(*Deactivate*)
ARsDeactivateDescription	[172]		:=		'[ DA-0172 ] OutputSignal - Reserved';
ARbDeactivateOutput		[172]		:=		FALSE or ARbDeactivateTestPB[172];

(*Deactivate*)
ARsDeactivateDescription	[173]		:=		'[ DA-0173 ] OutputSignal - Reserved';
ARbDeactivateOutput		[173]		:=		FALSE or ARbDeactivateTestPB[173];

(*Deactivate*)
ARsDeactivateDescription	[174]		:=		'[ DA-0174 ] OutputSignal - Reserved';
ARbDeactivateOutput		[174]		:=		FALSE or ARbDeactivateTestPB[174];

(*Deactivate*)
ARsDeactivateDescription	[175]		:=		'[ DA-0175 ] OutputSignal - Reserved';
ARbDeactivateOutput		[175]		:=		FALSE or ARbDeactivateTestPB[175];

(*Deactivate*)
ARsDeactivateDescription	[176]		:=		'[ DA-0176 ] OutputSignal - Reserved';
ARbDeactivateOutput		[176]		:=		FALSE or ARbDeactivateTestPB[176];

(*Deactivate*)
ARsDeactivateDescription	[177]		:=		'[ DA-0177 ] OutputSignal - Reserved';
ARbDeactivateOutput		[177]		:=		FALSE or ARbDeactivateTestPB[177];

(*Deactivate*)
ARsDeactivateDescription	[178]		:=		'[ DA-0178 ] OutputSignal - Reserved';
ARbDeactivateOutput		[178]		:=		FALSE or ARbDeactivateTestPB[178];

(*Deactivate*)
ARsDeactivateDescription	[179]		:=		'[ DA-0179 ] OutputSignal - Reserved';
ARbDeactivateOutput		[179]		:=		FALSE or ARbDeactivateTestPB[179];

(*Deactivate*)
ARsDeactivateDescription	[180]		:=		'[ DA-0180 ] OutputSignal - Reserved';
ARbDeactivateOutput		[180]		:=		FALSE or ARbDeactivateTestPB[180];

(*Deactivate*)
ARsDeactivateDescription	[181]		:=		'[ DA-0181 ] OutputSignal - Reserved';
ARbDeactivateOutput		[181]		:=		FALSE or ARbDeactivateTestPB[181];

(*Deactivate*)
ARsDeactivateDescription	[182]		:=		'[ DA-0182 ] OutputSignal - Reserved';
ARbDeactivateOutput		[182]		:=		FALSE or ARbDeactivateTestPB[182];

(*Deactivate*)
ARsDeactivateDescription	[183]		:=		'[ DA-0183 ] OutputSignal - Reserved';
ARbDeactivateOutput		[183]		:=		FALSE or ARbDeactivateTestPB[183];

(*Deactivate*)
ARsDeactivateDescription	[184]		:=		'[ DA-0184 ] OutputSignal - Reserved';
ARbDeactivateOutput		[184]		:=		FALSE or ARbDeactivateTestPB[184];

(*Deactivate*)
ARsDeactivateDescription	[185]		:=		'[ DA-0185 ] OutputSignal - Reserved';
ARbDeactivateOutput		[185]		:=		FALSE or ARbDeactivateTestPB[185];

(*Deactivate*)
ARsDeactivateDescription	[186]		:=		'[ DA-0186 ] OutputSignal - Reserved';
ARbDeactivateOutput		[186]		:=		FALSE or ARbDeactivateTestPB[186];

(*Deactivate*)
ARsDeactivateDescription	[187]		:=		'[ DA-0187 ] OutputSignal - Reserved';
ARbDeactivateOutput		[187]		:=		FALSE or ARbDeactivateTestPB[187];

(*Deactivate*)
ARsDeactivateDescription	[188]		:=		'[ DA-0188 ] OutputSignal - Reserved';
ARbDeactivateOutput		[188]		:=		FALSE or ARbDeactivateTestPB[188];

(*Deactivate*)
ARsDeactivateDescription	[189]		:=		'[ DA-0189 ] OutputSignal - Reserved';
ARbDeactivateOutput		[189]		:=		FALSE or ARbDeactivateTestPB[189];

(*Deactivate*)
ARsDeactivateDescription	[190]		:=		'[ DA-0190 ] OutputSignal - Reserved';
ARbDeactivateOutput		[190]		:=		FALSE or ARbDeactivateTestPB[190];

(*Deactivate*)
ARsDeactivateDescription	[191]		:=		'[ DA-0191 ] OutputSignal - Reserved';
ARbDeactivateOutput		[191]		:=		FALSE or ARbDeactivateTestPB[191];

(*Deactivate*)
ARsDeactivateDescription	[192]		:=		'[ DA-0192 ] OutputSignal - Reserved';
ARbDeactivateOutput		[192]		:=		FALSE or ARbDeactivateTestPB[192];

(*Deactivate*)
ARsDeactivateDescription	[193]		:=		'[ DA-0193 ] OutputSignal - Reserved';
ARbDeactivateOutput		[193]		:=		FALSE or ARbDeactivateTestPB[193];

(*Deactivate*)
ARsDeactivateDescription	[194]		:=		'[ DA-0194 ] OutputSignal - Reserved';
ARbDeactivateOutput		[194]		:=		FALSE or ARbDeactivateTestPB[194];

(*Deactivate*)
ARsDeactivateDescription	[195]		:=		'[ DA-0195 ] OutputSignal - Reserved';
ARbDeactivateOutput		[195]		:=		FALSE or ARbDeactivateTestPB[195];

(*Deactivate*)
ARsDeactivateDescription	[196]		:=		'[ DA-0196 ] OutputSignal - Reserved';
ARbDeactivateOutput		[196]		:=		FALSE or ARbDeactivateTestPB[196];

(*Deactivate*)
ARsDeactivateDescription	[197]		:=		'[ DA-0197 ] OutputSignal - Reserved';
ARbDeactivateOutput		[197]		:=		FALSE or ARbDeactivateTestPB[197];

(*Deactivate*)
ARsDeactivateDescription	[198]		:=		'[ DA-0198 ] OutputSignal - Reserved';
ARbDeactivateOutput		[198]		:=		FALSE or ARbDeactivateTestPB[198];

(*Deactivate*)
ARsDeactivateDescription	[199]		:=		'[ DA-0199 ] OutputSignal - Reserved';
ARbDeactivateOutput		[199]		:=		FALSE or ARbDeactivateTestPB[199];

(*Deactivate*)
ARsDeactivateDescription	[200]		:=		'[ DA-0200 ] OutputSignal - Reserved';
ARbDeactivateOutput		[200]		:=		FALSE or ARbDeactivateTestPB[200];
*)
*)

END_PROGRAM

// ---- POUs/MainProgram/AutoArmCtrl/OmronServoEnable.TcPOU
PROGRAM OmronServoEnable
VAR
END_VAR

IF PowerOnDelay.Q AND NOT EmergencyStop THEN
	ARwDO[eY10007_STN09SLOWPULLMECHANISMSERVOMOTOR_ERRORSTOP].00 := TRUE;
	ARwDO[eY10008_Arm01HorizontalServoMotor_ErrorStop].00 := TRUE;
	ARwDO[eY10009_Arm01VerticalServoMotor_ErrorStop].00 := TRUE;
	ELSE
	ARwDO[eY10007_STN09SLOWPULLMECHANISMSERVOMOTOR_ERRORSTOP].00 := FALSE;
	ARwDO[eY10008_Arm01HorizontalServoMotor_ErrorStop].00 := FALSE;
	ARwDO[eY10009_Arm01VerticalServoMotor_ErrorStop].00 := FALSE;
END_IF

END_PROGRAM

// ---- POUs/MainProgram/AutoArmCtrl/AxisHorzMovementOutputCtrl_Arm1.TcPOU
PROGRAM AxisHorzMovementOutputCtrl_Arm1
VAR

	LdUnhook: CMP_OC_DW;
	Stn1Unhook: CMP_OC_DW;
	Stn2Unhook: CMP_OC_DW;
	Stn3Unhook: CMP_OC_DW;
	Stn4Unhook: CMP_OC_DW;
	Stn5Unhook: CMP_OC_DW;
	Stn6Unhook: CMP_OC_DW;
	Stn7Unhook: CMP_OC_DW;
	Stn8Unhook: CMP_OC_DW;
	Stn9Unhook: CMP_OC_DW;
	Stn10Unhook: CMP_OC_DW;
	Stn11Unhook: CMP_OC_DW;
	Stn12Unhook: CMP_OC_DW;
	Uld1Unhook: CMP_OC_DW;
	Uld2Unhook: CMP_OC_DW;

	LdHook: CMP_OC_DW;
	Stn1Hook: CMP_OC_DW;
	Stn2Hook: CMP_OC_DW;
	Stn3Hook: CMP_OC_DW;
	Stn4Hook: CMP_OC_DW;
	Stn5Hook: CMP_OC_DW;
	Stn6Hook: CMP_OC_DW;
	Stn7Hook: CMP_OC_DW;
	Stn8Hook: CMP_OC_DW;
	Stn9Hook: CMP_OC_DW;
	Stn10Hook: CMP_OC_DW;
	Stn11Hook: CMP_OC_DW;
	Stn12Hook: CMP_OC_DW;
	Uld1Hook: CMP_OC_DW;
	Uld2Hook: CMP_OC_DW;

END_VAR

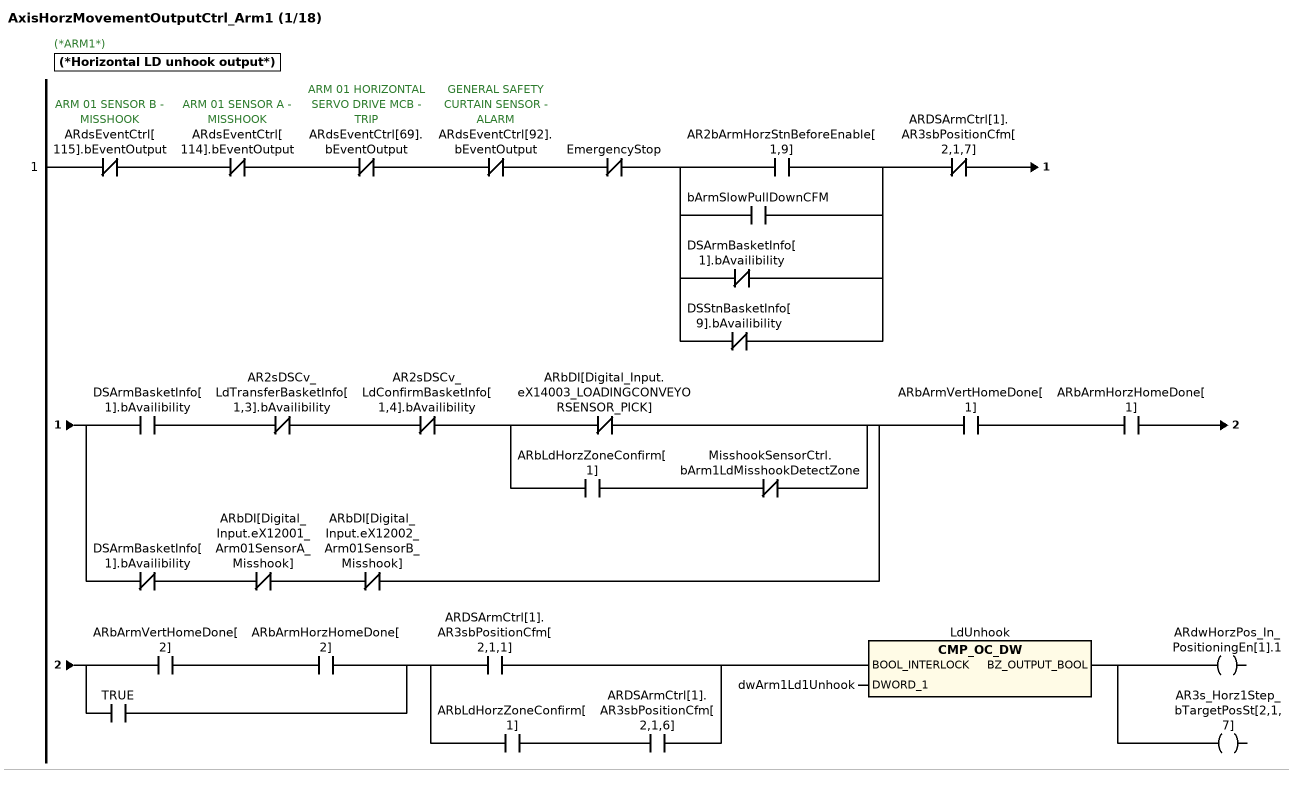
// NETWORK 1
// (*ARM1*)
//   ARdsEventCtrl[115].bEventOutput: ARM 01 SENSOR B - MISSHOOK
//   ARdsEventCtrl[114].bEventOutput: ARM 01 SENSOR A - MISSHOOK
//   ARdsEventCtrl[69].bEventOutput: ARM 01 HORIZONTAL SERVO DRIVE MCB - TRIP
//   ARdsEventCtrl[92].bEventOutput: GENERAL SAFETY CURTAIN SENSOR - ALARM
// label: (*Horizontal LD unhook output*)
LdUnhook(BOOL_INTERLOCK := (((NOT ARdsEventCtrl[115].bEventOutput AND NOT ARdsEventCtrl[114].bEventOutput AND NOT ARdsEventCtrl[69].bEventOutput AND NOT ARdsEventCtrl[92].bEventOutput AND NOT EmergencyStop) AND (AR2bArmHorzStnBeforeEnable[1,9] OR bArmSlowPullDownCFM OR NOT DSArmBasketInfo[1].bAvailibility OR NOT DSStnBasketInfo[9].bAvailibility)) AND NOT ARDSArmCtrl[1].AR3sbPositionCfm[2,1,7] AND (DSArmBasketInfo[1].bAvailibility AND NOT AR2sDSCv_LdTransferBasketInfo[1,3].bAvailibility AND NOT AR2sDSCv_LdConfirmBasketInfo[1,4].bAvailibility AND (NOT ARbDI[Digital_Input.eX14003_LOADINGCONVEYORSENSOR_PICK] OR ARbLdHorzZoneConfirm[1] AND NOT MisshookSensorCtrl.bArm1LdMisshookDetectZone) OR NOT DSArmBasketInfo[1].bAvailibility AND NOT ARbDI[Digital_Input.eX12001_Arm01SensorA_Misshook] AND NOT ARbDI[Digital_Input.eX12002_Arm01SensorB_Misshook])) AND ARbArmVertHomeDone[1] AND ARbArmHorzHomeDone[1] AND (ARbArmVertHomeDone[2] AND ARbArmHorzHomeDone[2] OR TRUE) AND (ARDSArmCtrl[1].AR3sbPositionCfm[2,1,1] OR ARbLdHorzZoneConfirm[1] AND ARDSArmCtrl[1].AR3sbPositionCfm[2,1,6]), DWORD_1 := dwArm1Ld1Unhook); // CMP_OC_DW
ARdwHorzPos_In_PositioningEn[1].1 := LdUnhook.BZ_OUTPUT_BOOL;
AR3s_Horz1Step_bTargetPosSt[2,1,7] := LdUnhook.BZ_OUTPUT_BOOL;

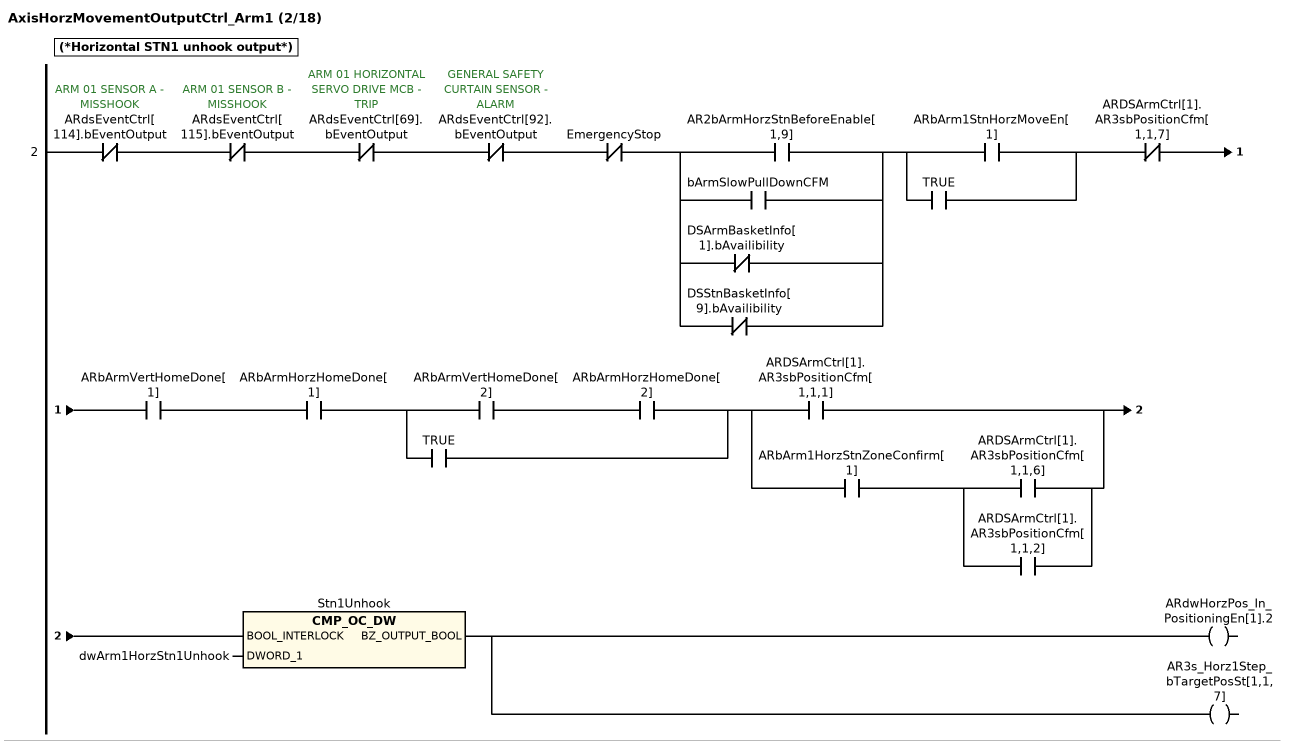
// NETWORK 2
//   ARdsEventCtrl[114].bEventOutput: ARM 01 SENSOR A - MISSHOOK
//   ARdsEventCtrl[115].bEventOutput: ARM 01 SENSOR B - MISSHOOK
//   ARdsEventCtrl[69].bEventOutput: ARM 01 HORIZONTAL SERVO DRIVE MCB - TRIP
//   ARdsEventCtrl[92].bEventOutput: GENERAL SAFETY CURTAIN SENSOR - ALARM
// label: (*Horizontal STN1 unhook output*)
Stn1Unhook(BOOL_INTERLOCK := ((NOT ARdsEventCtrl[114].bEventOutput AND NOT ARdsEventCtrl[115].bEventOutput AND NOT ARdsEventCtrl[69].bEventOutput AND NOT ARdsEventCtrl[92].bEventOutput AND NOT EmergencyStop) AND (AR2bArmHorzStnBeforeEnable[1,9] OR bArmSlowPullDownCFM OR NOT DSArmBasketInfo[1].bAvailibility OR NOT DSStnBasketInfo[9].bAvailibility) AND (ARbArm1StnHorzMoveEn[1] OR TRUE)) AND NOT ARDSArmCtrl[1].AR3sbPositionCfm[1,1,7] AND ARbArmVertHomeDone[1] AND ARbArmHorzHomeDone[1] AND (ARbArmVertHomeDone[2] AND ARbArmHorzHomeDone[2] OR TRUE) AND (ARDSArmCtrl[1].AR3sbPositionCfm[1,1,1] OR ARbArm1HorzStnZoneConfirm[1] AND (ARDSArmCtrl[1].AR3sbPositionCfm[1,1,6] OR ARDSArmCtrl[1].AR3sbPositionCfm[1,1,2])), DWORD_1 := dwArm1HorzStn1Unhook); // CMP_OC_DW
ARdwHorzPos_In_PositioningEn[1].2 := Stn1Unhook.BZ_OUTPUT_BOOL;
AR3s_Horz1Step_bTargetPosSt[1,1,7] := Stn1Unhook.BZ_OUTPUT_BOOL;

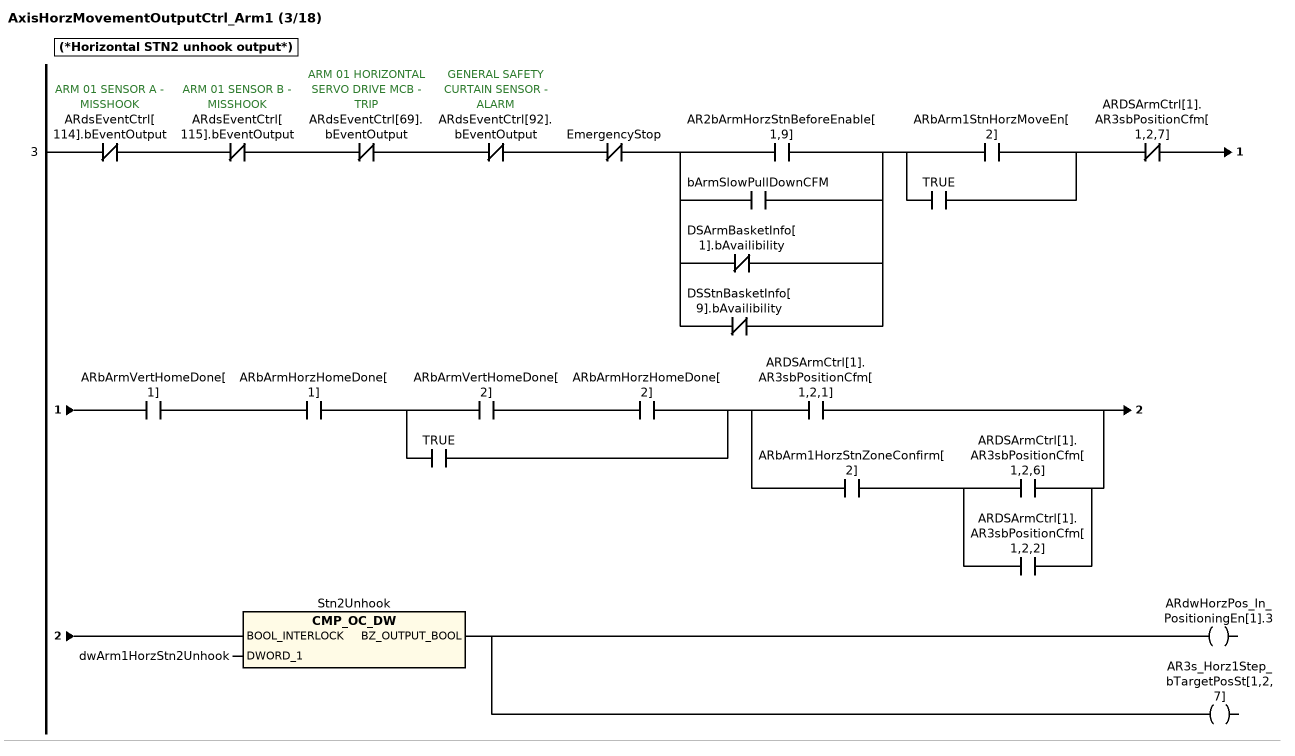
// NETWORK 3
//   ARdsEventCtrl[114].bEventOutput: ARM 01 SENSOR A - MISSHOOK
//   ARdsEventCtrl[115].bEventOutput: ARM 01 SENSOR B - MISSHOOK
//   ARdsEventCtrl[69].bEventOutput: ARM 01 HORIZONTAL SERVO DRIVE MCB - TRIP
//   ARdsEventCtrl[92].bEventOutput: GENERAL SAFETY CURTAIN SENSOR - ALARM
// label: (*Horizontal STN2 unhook output*)
Stn2Unhook(BOOL_INTERLOCK := ((NOT ARdsEventCtrl[114].bEventOutput AND NOT ARdsEventCtrl[115].bEventOutput AND NOT ARdsEventCtrl[69].bEventOutput AND NOT ARdsEventCtrl[92].bEventOutput AND NOT EmergencyStop) AND (AR2bArmHorzStnBeforeEnable[1,9] OR bArmSlowPullDownCFM OR NOT DSArmBasketInfo[1].bAvailibility OR NOT DSStnBasketInfo[9].bAvailibility) AND (ARbArm1StnHorzMoveEn[2] OR TRUE)) AND NOT ARDSArmCtrl[1].AR3sbPositionCfm[1,2,7] AND ARbArmVertHomeDone[1] AND ARbArmHorzHomeDone[1] AND (ARbArmVertHomeDone[2] AND ARbArmHorzHomeDone[2] OR TRUE) AND (ARDSArmCtrl[1].AR3sbPositionCfm[1,2,1] OR ARbArm1HorzStnZoneConfirm[2] AND (ARDSArmCtrl[1].AR3sbPositionCfm[1,2,6] OR ARDSArmCtrl[1].AR3sbPositionCfm[1,2,2])), DWORD_1 := dwArm1HorzStn2Unhook); // CMP_OC_DW
ARdwHorzPos_In_PositioningEn[1].3 := Stn2Unhook.BZ_OUTPUT_BOOL;
AR3s_Horz1Step_bTargetPosSt[1,2,7] := Stn2Unhook.BZ_OUTPUT_BOOL;

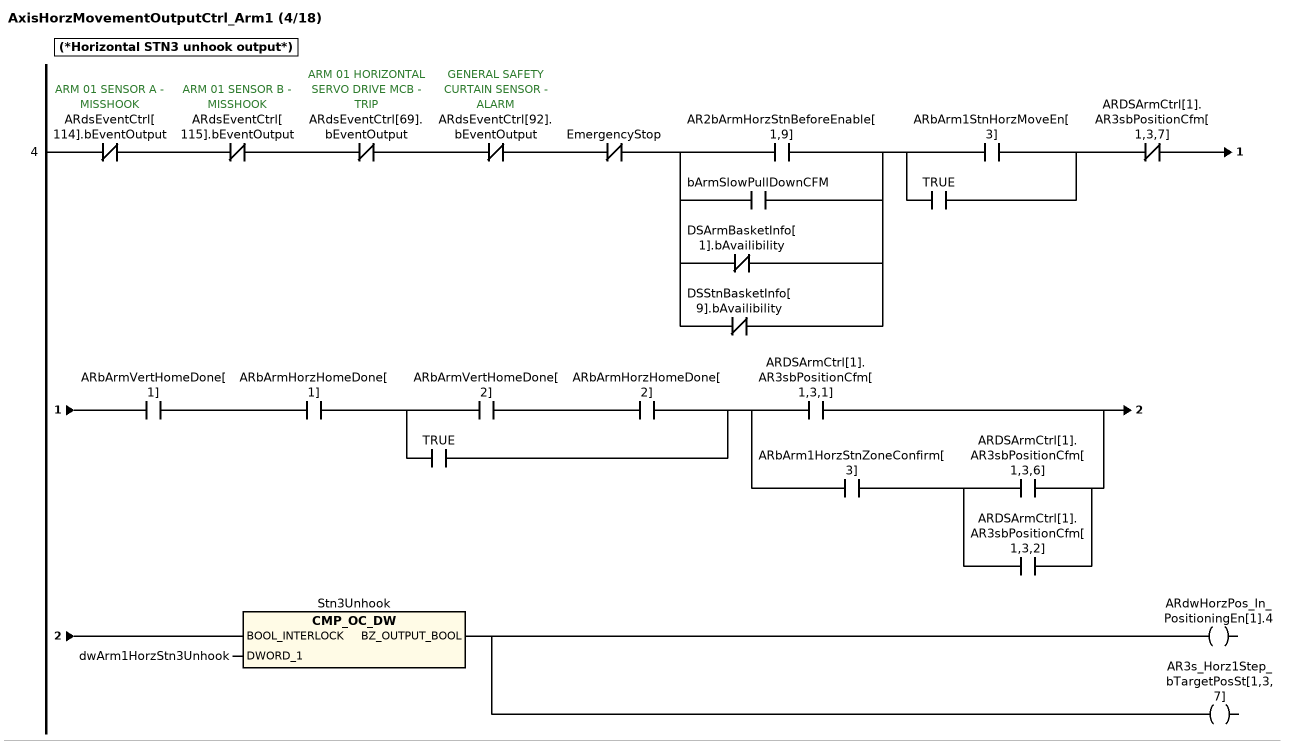
// NETWORK 4
//   ARdsEventCtrl[114].bEventOutput: ARM 01 SENSOR A - MISSHOOK
//   ARdsEventCtrl[115].bEventOutput: ARM 01 SENSOR B - MISSHOOK
//   ARdsEventCtrl[69].bEventOutput: ARM 01 HORIZONTAL SERVO DRIVE MCB - TRIP
//   ARdsEventCtrl[92].bEventOutput: GENERAL SAFETY CURTAIN SENSOR - ALARM
// label: (*Horizontal STN3 unhook output*)
Stn3Unhook(BOOL_INTERLOCK := ((NOT ARdsEventCtrl[114].bEventOutput AND NOT ARdsEventCtrl[115].bEventOutput AND NOT ARdsEventCtrl[69].bEventOutput AND NOT ARdsEventCtrl[92].bEventOutput AND NOT EmergencyStop) AND (AR2bArmHorzStnBeforeEnable[1,9] OR bArmSlowPullDownCFM OR NOT DSArmBasketInfo[1].bAvailibility OR NOT DSStnBasketInfo[9].bAvailibility) AND (ARbArm1StnHorzMoveEn[3] OR TRUE)) AND NOT ARDSArmCtrl[1].AR3sbPositionCfm[1,3,7] AND ARbArmVertHomeDone[1] AND ARbArmHorzHomeDone[1] AND (ARbArmVertHomeDone[2] AND ARbArmHorzHomeDone[2] OR TRUE) AND (ARDSArmCtrl[1].AR3sbPositionCfm[1,3,1] OR ARbArm1HorzStnZoneConfirm[3] AND (ARDSArmCtrl[1].AR3sbPositionCfm[1,3,6] OR ARDSArmCtrl[1].AR3sbPositionCfm[1,3,2])), DWORD_1 := dwArm1HorzStn3Unhook); // CMP_OC_DW
ARdwHorzPos_In_PositioningEn[1].4 := Stn3Unhook.BZ_OUTPUT_BOOL;
AR3s_Horz1Step_bTargetPosSt[1,3,7] := Stn3Unhook.BZ_OUTPUT_BOOL;

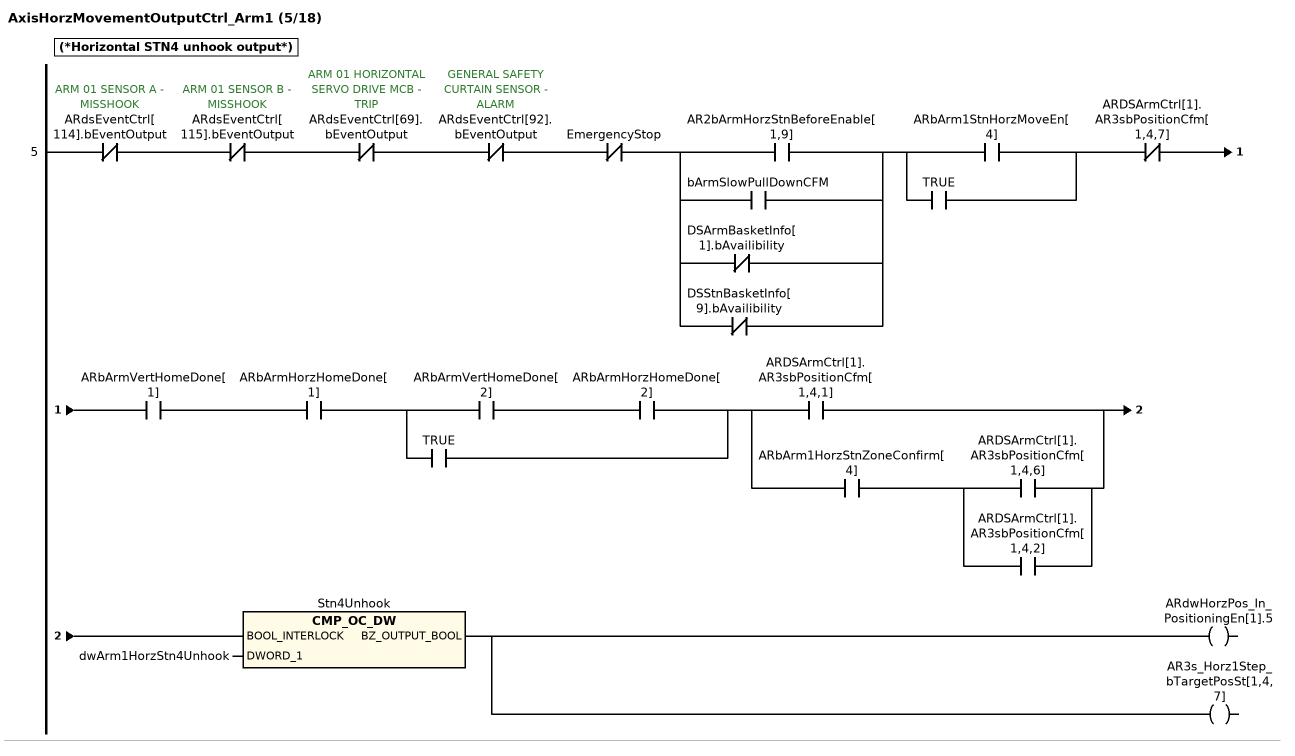
// NETWORK 5
//   ARdsEventCtrl[114].bEventOutput: ARM 01 SENSOR A - MISSHOOK
//   ARdsEventCtrl[115].bEventOutput: ARM 01 SENSOR B - MISSHOOK
//   ARdsEventCtrl[69].bEventOutput: ARM 01 HORIZONTAL SERVO DRIVE MCB - TRIP
//   ARdsEventCtrl[92].bEventOutput: GENERAL SAFETY CURTAIN SENSOR - ALARM
// label: (*Horizontal STN4 unhook output*)
Stn4Unhook(BOOL_INTERLOCK := ((NOT ARdsEventCtrl[114].bEventOutput AND NOT ARdsEventCtrl[115].bEventOutput AND NOT ARdsEventCtrl[69].bEventOutput AND NOT ARdsEventCtrl[92].bEventOutput AND NOT EmergencyStop) AND (AR2bArmHorzStnBeforeEnable[1,9] OR bArmSlowPullDownCFM OR NOT DSArmBasketInfo[1].bAvailibility OR NOT DSStnBasketInfo[9].bAvailibility) AND (ARbArm1StnHorzMoveEn[4] OR TRUE)) AND NOT ARDSArmCtrl[1].AR3sbPositionCfm[1,4,7] AND ARbArmVertHomeDone[1] AND ARbArmHorzHomeDone[1] AND (ARbArmVertHomeDone[2] AND ARbArmHorzHomeDone[2] OR TRUE) AND (ARDSArmCtrl[1].AR3sbPositionCfm[1,4,1] OR ARbArm1HorzStnZoneConfirm[4] AND (ARDSArmCtrl[1].AR3sbPositionCfm[1,4,6] OR ARDSArmCtrl[1].AR3sbPositionCfm[1,4,2])), DWORD_1 := dwArm1HorzStn4Unhook); // CMP_OC_DW
ARdwHorzPos_In_PositioningEn[1].5 := Stn4Unhook.BZ_OUTPUT_BOOL;
AR3s_Horz1Step_bTargetPosSt[1,4,7] := Stn4Unhook.BZ_OUTPUT_BOOL;

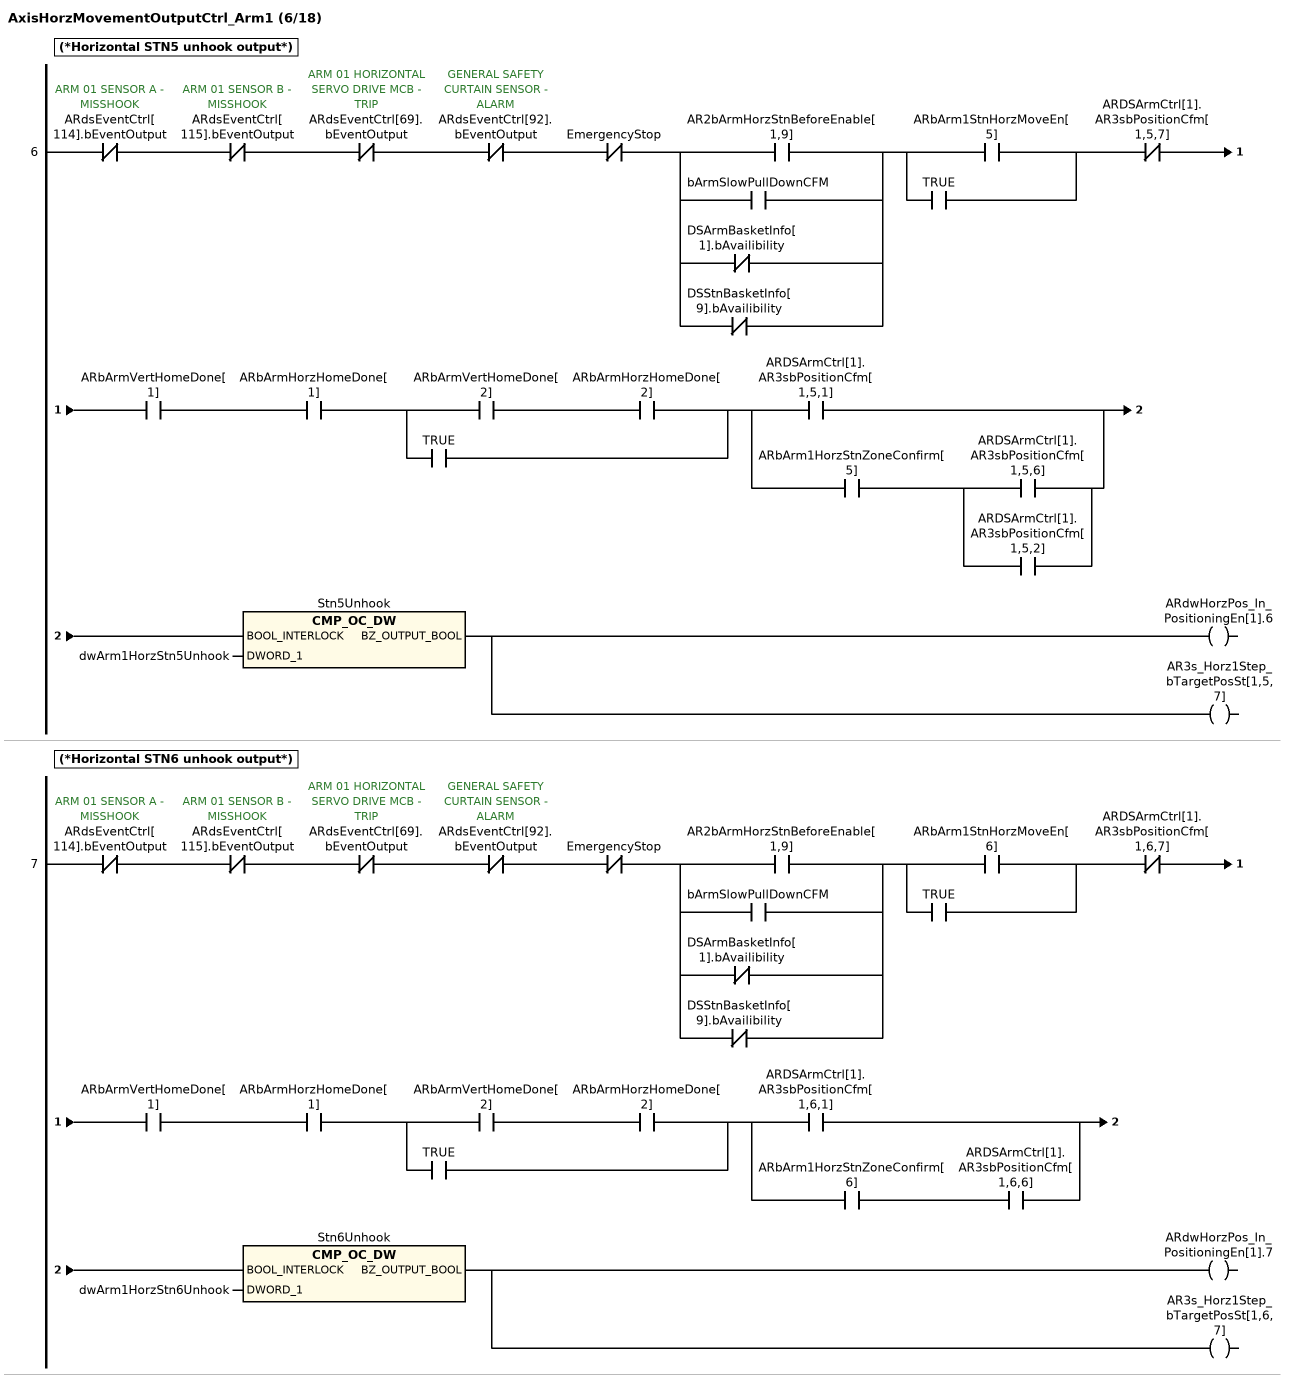
// NETWORK 6
//   ARdsEventCtrl[114].bEventOutput: ARM 01 SENSOR A - MISSHOOK
//   ARdsEventCtrl[115].bEventOutput: ARM 01 SENSOR B - MISSHOOK
//   ARdsEventCtrl[69].bEventOutput: ARM 01 HORIZONTAL SERVO DRIVE MCB - TRIP
//   ARdsEventCtrl[92].bEventOutput: GENERAL SAFETY CURTAIN SENSOR - ALARM
// label: (*Horizontal STN5 unhook output*)
Stn5Unhook(BOOL_INTERLOCK := ((NOT ARdsEventCtrl[114].bEventOutput AND NOT ARdsEventCtrl[115].bEventOutput AND NOT ARdsEventCtrl[69].bEventOutput AND NOT ARdsEventCtrl[92].bEventOutput AND NOT EmergencyStop) AND (AR2bArmHorzStnBeforeEnable[1,9] OR bArmSlowPullDownCFM OR NOT DSArmBasketInfo[1].bAvailibility OR NOT DSStnBasketInfo[9].bAvailibility) AND (ARbArm1StnHorzMoveEn[5] OR TRUE)) AND NOT ARDSArmCtrl[1].AR3sbPositionCfm[1,5,7] AND ARbArmVertHomeDone[1] AND ARbArmHorzHomeDone[1] AND (ARbArmVertHomeDone[2] AND ARbArmHorzHomeDone[2] OR TRUE) AND (ARDSArmCtrl[1].AR3sbPositionCfm[1,5,1] OR ARbArm1HorzStnZoneConfirm[5] AND (ARDSArmCtrl[1].AR3sbPositionCfm[1,5,6] OR ARDSArmCtrl[1].AR3sbPositionCfm[1,5,2])), DWORD_1 := dwArm1HorzStn5Unhook); // CMP_OC_DW
ARdwHorzPos_In_PositioningEn[1].6 := Stn5Unhook.BZ_OUTPUT_BOOL;
AR3s_Horz1Step_bTargetPosSt[1,5,7] := Stn5Unhook.BZ_OUTPUT_BOOL;

// NETWORK 7
//   ARdsEventCtrl[114].bEventOutput: ARM 01 SENSOR A - MISSHOOK
//   ARdsEventCtrl[115].bEventOutput: ARM 01 SENSOR B - MISSHOOK
//   ARdsEventCtrl[69].bEventOutput: ARM 01 HORIZONTAL SERVO DRIVE MCB - TRIP
//   ARdsEventCtrl[92].bEventOutput: GENERAL SAFETY CURTAIN SENSOR - ALARM
// label: (*Horizontal STN6 unhook output*)
Stn6Unhook(BOOL_INTERLOCK := ((NOT ARdsEventCtrl[114].bEventOutput AND NOT ARdsEventCtrl[115].bEventOutput AND NOT ARdsEventCtrl[69].bEventOutput AND NOT ARdsEventCtrl[92].bEventOutput AND NOT EmergencyStop) AND ((AR2bArmHorzStnBeforeEnable[1,9] OR bArmSlowPullDownCFM OR NOT DSArmBasketInfo[1].bAvailibility OR NOT DSStnBasketInfo[9].bAvailibility) AND (ARbArm1StnHorzMoveEn[6] OR TRUE))) AND NOT ARDSArmCtrl[1].AR3sbPositionCfm[1,6,7] AND ARbArmVertHomeDone[1] AND ARbArmHorzHomeDone[1] AND (ARbArmVertHomeDone[2] AND ARbArmHorzHomeDone[2] OR TRUE) AND (ARDSArmCtrl[1].AR3sbPositionCfm[1,6,1] OR ARbArm1HorzStnZoneConfirm[6] AND ARDSArmCtrl[1].AR3sbPositionCfm[1,6,6]), DWORD_1 := dwArm1HorzStn6Unhook); // CMP_OC_DW
ARdwHorzPos_In_PositioningEn[1].7 := Stn6Unhook.BZ_OUTPUT_BOOL;
AR3s_Horz1Step_bTargetPosSt[1,6,7] := Stn6Unhook.BZ_OUTPUT_BOOL;

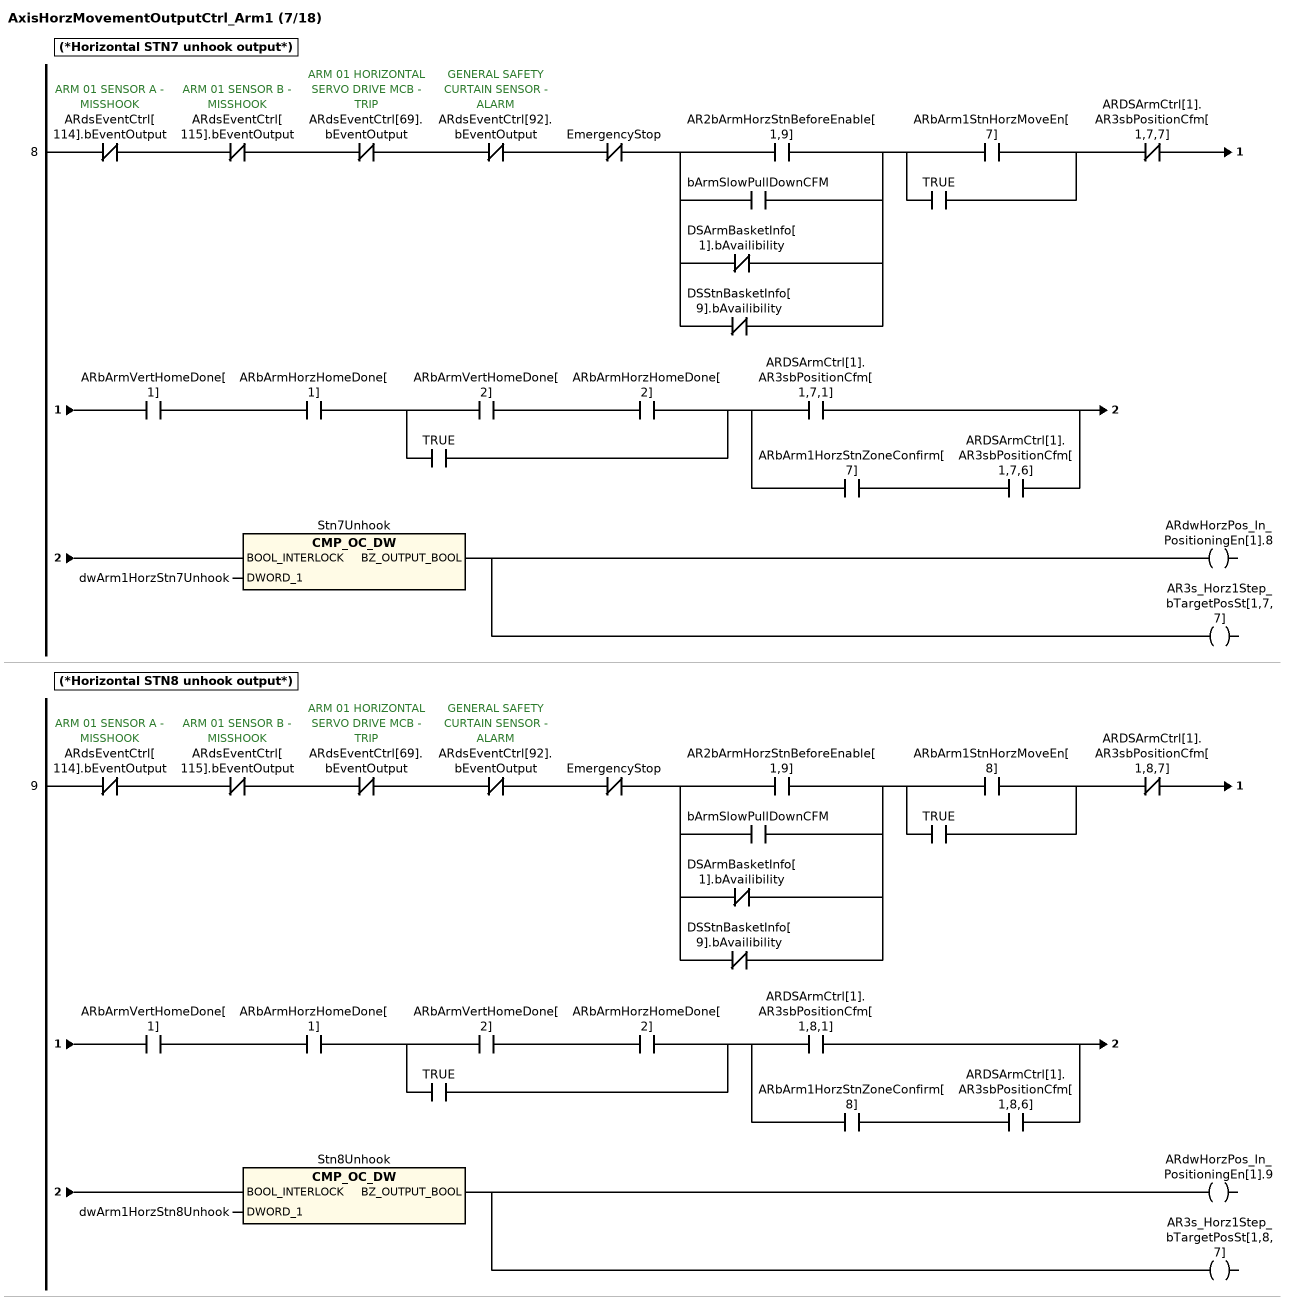
// NETWORK 8
//   ARdsEventCtrl[114].bEventOutput: ARM 01 SENSOR A - MISSHOOK
//   ARdsEventCtrl[115].bEventOutput: ARM 01 SENSOR B - MISSHOOK
//   ARdsEventCtrl[69].bEventOutput: ARM 01 HORIZONTAL SERVO DRIVE MCB - TRIP
//   ARdsEventCtrl[92].bEventOutput: GENERAL SAFETY CURTAIN SENSOR - ALARM
// label: (*Horizontal STN7 unhook output*)
Stn7Unhook(BOOL_INTERLOCK := ((NOT ARdsEventCtrl[114].bEventOutput AND NOT ARdsEventCtrl[115].bEventOutput AND NOT ARdsEventCtrl[69].bEventOutput AND NOT ARdsEventCtrl[92].bEventOutput AND NOT EmergencyStop) AND (AR2bArmHorzStnBeforeEnable[1,9] OR bArmSlowPullDownCFM OR NOT DSArmBasketInfo[1].bAvailibility OR NOT DSStnBasketInfo[9].bAvailibility) AND (ARbArm1StnHorzMoveEn[7] OR TRUE)) AND NOT ARDSArmCtrl[1].AR3sbPositionCfm[1,7,7] AND ARbArmVertHomeDone[1] AND ARbArmHorzHomeDone[1] AND (ARbArmVertHomeDone[2] AND ARbArmHorzHomeDone[2] OR TRUE) AND (ARDSArmCtrl[1].AR3sbPositionCfm[1,7,1] OR ARbArm1HorzStnZoneConfirm[7] AND ARDSArmCtrl[1].AR3sbPositionCfm[1,7,6]), DWORD_1 := dwArm1HorzStn7Unhook); // CMP_OC_DW
ARdwHorzPos_In_PositioningEn[1].8 := Stn7Unhook.BZ_OUTPUT_BOOL;
AR3s_Horz1Step_bTargetPosSt[1,7,7] := Stn7Unhook.BZ_OUTPUT_BOOL;

// NETWORK 9
//   ARdsEventCtrl[114].bEventOutput: ARM 01 SENSOR A - MISSHOOK
//   ARdsEventCtrl[115].bEventOutput: ARM 01 SENSOR B - MISSHOOK
//   ARdsEventCtrl[69].bEventOutput: ARM 01 HORIZONTAL SERVO DRIVE MCB - TRIP
//   ARdsEventCtrl[92].bEventOutput: GENERAL SAFETY CURTAIN SENSOR - ALARM
// label: (*Horizontal STN8 unhook output*)
Stn8Unhook(BOOL_INTERLOCK := ((NOT ARdsEventCtrl[114].bEventOutput AND NOT ARdsEventCtrl[115].bEventOutput AND NOT ARdsEventCtrl[69].bEventOutput AND NOT ARdsEventCtrl[92].bEventOutput AND NOT EmergencyStop) AND (AR2bArmHorzStnBeforeEnable[1,9] OR bArmSlowPullDownCFM OR NOT DSArmBasketInfo[1].bAvailibility OR NOT DSStnBasketInfo[9].bAvailibility) AND (ARbArm1StnHorzMoveEn[8] OR TRUE)) AND NOT ARDSArmCtrl[1].AR3sbPositionCfm[1,8,7] AND ARbArmVertHomeDone[1] AND ARbArmHorzHomeDone[1] AND (ARbArmVertHomeDone[2] AND ARbArmHorzHomeDone[2] OR TRUE) AND (ARDSArmCtrl[1].AR3sbPositionCfm[1,8,1] OR ARbArm1HorzStnZoneConfirm[8] AND ARDSArmCtrl[1].AR3sbPositionCfm[1,8,6]), DWORD_1 := dwArm1HorzStn8Unhook); // CMP_OC_DW
ARdwHorzPos_In_PositioningEn[1].9 := Stn8Unhook.BZ_OUTPUT_BOOL;
AR3s_Horz1Step_bTargetPosSt[1,8,7] := Stn8Unhook.BZ_OUTPUT_BOOL;

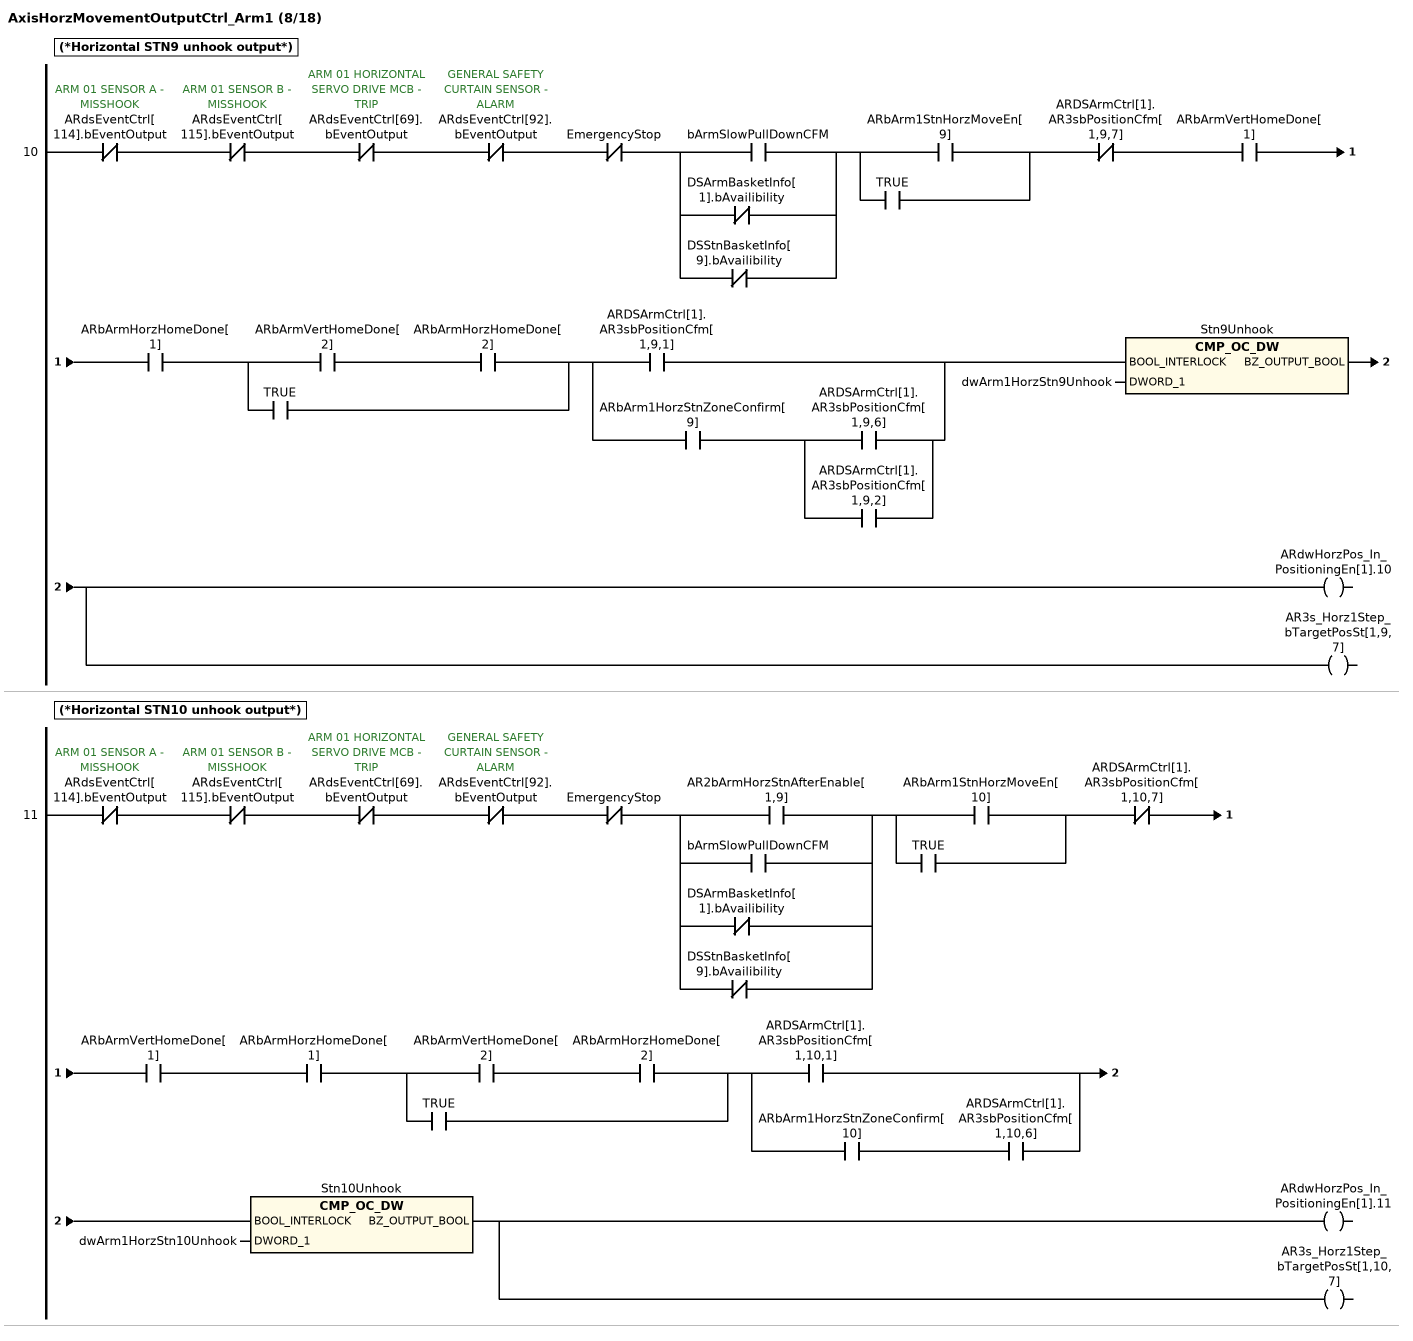
// NETWORK 10
//   ARdsEventCtrl[114].bEventOutput: ARM 01 SENSOR A - MISSHOOK
//   ARdsEventCtrl[115].bEventOutput: ARM 01 SENSOR B - MISSHOOK
//   ARdsEventCtrl[69].bEventOutput: ARM 01 HORIZONTAL SERVO DRIVE MCB - TRIP
//   ARdsEventCtrl[92].bEventOutput: GENERAL SAFETY CURTAIN SENSOR - ALARM
// label: (*Horizontal STN9 unhook output*)
Stn9Unhook(BOOL_INTERLOCK := ((NOT ARdsEventCtrl[114].bEventOutput AND NOT ARdsEventCtrl[115].bEventOutput AND NOT ARdsEventCtrl[69].bEventOutput AND NOT ARdsEventCtrl[92].bEventOutput AND NOT EmergencyStop) AND (bArmSlowPullDownCFM OR NOT DSArmBasketInfo[1].bAvailibility OR NOT DSStnBasketInfo[9].bAvailibility) AND (ARbArm1StnHorzMoveEn[9] OR TRUE)) AND NOT ARDSArmCtrl[1].AR3sbPositionCfm[1,9,7] AND ARbArmVertHomeDone[1] AND ARbArmHorzHomeDone[1] AND (ARbArmVertHomeDone[2] AND ARbArmHorzHomeDone[2] OR TRUE) AND (ARDSArmCtrl[1].AR3sbPositionCfm[1,9,1] OR ARbArm1HorzStnZoneConfirm[9] AND (ARDSArmCtrl[1].AR3sbPositionCfm[1,9,6] OR ARDSArmCtrl[1].AR3sbPositionCfm[1,9,2])), DWORD_1 := dwArm1HorzStn9Unhook); // CMP_OC_DW
ARdwHorzPos_In_PositioningEn[1].10 := Stn9Unhook.BZ_OUTPUT_BOOL;
AR3s_Horz1Step_bTargetPosSt[1,9,7] := Stn9Unhook.BZ_OUTPUT_BOOL;

// NETWORK 11
//   ARdsEventCtrl[114].bEventOutput: ARM 01 SENSOR A - MISSHOOK
//   ARdsEventCtrl[115].bEventOutput: ARM 01 SENSOR B - MISSHOOK
//   ARdsEventCtrl[69].bEventOutput: ARM 01 HORIZONTAL SERVO DRIVE MCB - TRIP
//   ARdsEventCtrl[92].bEventOutput: GENERAL SAFETY CURTAIN SENSOR - ALARM
// label: (*Horizontal STN10 unhook output*)
Stn10Unhook(BOOL_INTERLOCK := ((NOT ARdsEventCtrl[114].bEventOutput AND NOT ARdsEventCtrl[115].bEventOutput AND NOT ARdsEventCtrl[69].bEventOutput AND NOT ARdsEventCtrl[92].bEventOutput AND NOT EmergencyStop) AND (AR2bArmHorzStnAfterEnable[1,9] OR bArmSlowPullDownCFM OR NOT DSArmBasketInfo[1].bAvailibility OR NOT DSStnBasketInfo[9].bAvailibility) AND (ARbArm1StnHorzMoveEn[10] OR TRUE)) AND NOT ARDSArmCtrl[1].AR3sbPositionCfm[1,10,7] AND ARbArmVertHomeDone[1] AND ARbArmHorzHomeDone[1] AND (ARbArmVertHomeDone[2] AND ARbArmHorzHomeDone[2] OR TRUE) AND (ARDSArmCtrl[1].AR3sbPositionCfm[1,10,1] OR ARbArm1HorzStnZoneConfirm[10] AND ARDSArmCtrl[1].AR3sbPositionCfm[1,10,6]), DWORD_1 := dwArm1HorzStn10Unhook); // CMP_OC_DW
ARdwHorzPos_In_PositioningEn[1].11 := Stn10Unhook.BZ_OUTPUT_BOOL;
AR3s_Horz1Step_bTargetPosSt[1,10,7] := Stn10Unhook.BZ_OUTPUT_BOOL;

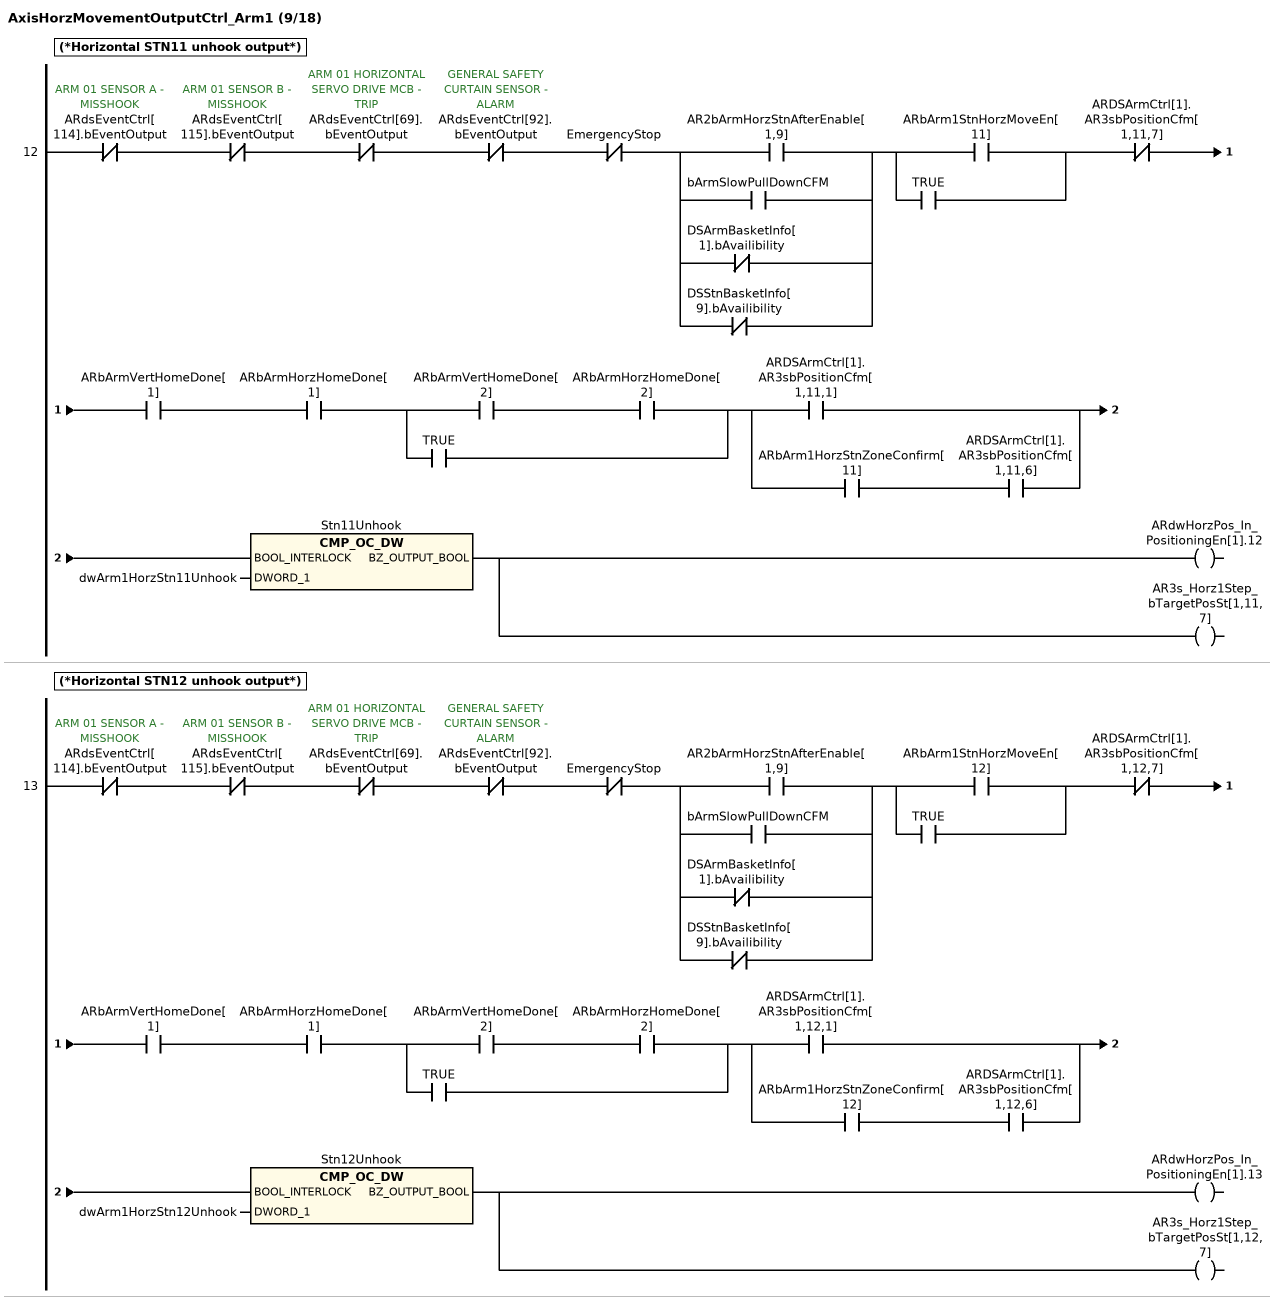
// NETWORK 12
//   ARdsEventCtrl[114].bEventOutput: ARM 01 SENSOR A - MISSHOOK
//   ARdsEventCtrl[115].bEventOutput: ARM 01 SENSOR B - MISSHOOK
//   ARdsEventCtrl[69].bEventOutput: ARM 01 HORIZONTAL SERVO DRIVE MCB - TRIP
//   ARdsEventCtrl[92].bEventOutput: GENERAL SAFETY CURTAIN SENSOR - ALARM
// label: (*Horizontal STN11 unhook output*)
Stn11Unhook(BOOL_INTERLOCK := ((NOT ARdsEventCtrl[114].bEventOutput AND NOT ARdsEventCtrl[115].bEventOutput AND NOT ARdsEventCtrl[69].bEventOutput AND NOT ARdsEventCtrl[92].bEventOutput AND NOT EmergencyStop) AND (AR2bArmHorzStnAfterEnable[1,9] OR bArmSlowPullDownCFM OR NOT DSArmBasketInfo[1].bAvailibility OR NOT DSStnBasketInfo[9].bAvailibility) AND (ARbArm1StnHorzMoveEn[11] OR TRUE)) AND NOT ARDSArmCtrl[1].AR3sbPositionCfm[1,11,7] AND ARbArmVertHomeDone[1] AND ARbArmHorzHomeDone[1] AND (ARbArmVertHomeDone[2] AND ARbArmHorzHomeDone[2] OR TRUE) AND (ARDSArmCtrl[1].AR3sbPositionCfm[1,11,1] OR ARbArm1HorzStnZoneConfirm[11] AND ARDSArmCtrl[1].AR3sbPositionCfm[1,11,6]), DWORD_1 := dwArm1HorzStn11Unhook); // CMP_OC_DW
ARdwHorzPos_In_PositioningEn[1].12 := Stn11Unhook.BZ_OUTPUT_BOOL;
AR3s_Horz1Step_bTargetPosSt[1,11,7] := Stn11Unhook.BZ_OUTPUT_BOOL;

// NETWORK 13
//   ARdsEventCtrl[114].bEventOutput: ARM 01 SENSOR A - MISSHOOK
//   ARdsEventCtrl[115].bEventOutput: ARM 01 SENSOR B - MISSHOOK
//   ARdsEventCtrl[69].bEventOutput: ARM 01 HORIZONTAL SERVO DRIVE MCB - TRIP
//   ARdsEventCtrl[92].bEventOutput: GENERAL SAFETY CURTAIN SENSOR - ALARM
// label: (*Horizontal STN12 unhook output*)
Stn12Unhook(BOOL_INTERLOCK := ((NOT ARdsEventCtrl[114].bEventOutput AND NOT ARdsEventCtrl[115].bEventOutput AND NOT ARdsEventCtrl[69].bEventOutput AND NOT ARdsEventCtrl[92].bEventOutput AND NOT EmergencyStop) AND (AR2bArmHorzStnAfterEnable[1,9] OR bArmSlowPullDownCFM OR NOT DSArmBasketInfo[1].bAvailibility OR NOT DSStnBasketInfo[9].bAvailibility) AND (ARbArm1StnHorzMoveEn[12] OR TRUE)) AND NOT ARDSArmCtrl[1].AR3sbPositionCfm[1,12,7] AND ARbArmVertHomeDone[1] AND ARbArmHorzHomeDone[1] AND (ARbArmVertHomeDone[2] AND ARbArmHorzHomeDone[2] OR TRUE) AND (ARDSArmCtrl[1].AR3sbPositionCfm[1,12,1] OR ARbArm1HorzStnZoneConfirm[12] AND ARDSArmCtrl[1].AR3sbPositionCfm[1,12,6]), DWORD_1 := dwArm1HorzStn12Unhook); // CMP_OC_DW
ARdwHorzPos_In_PositioningEn[1].13 := Stn12Unhook.BZ_OUTPUT_BOOL;
AR3s_Horz1Step_bTargetPosSt[1,12,7] := Stn12Unhook.BZ_OUTPUT_BOOL;

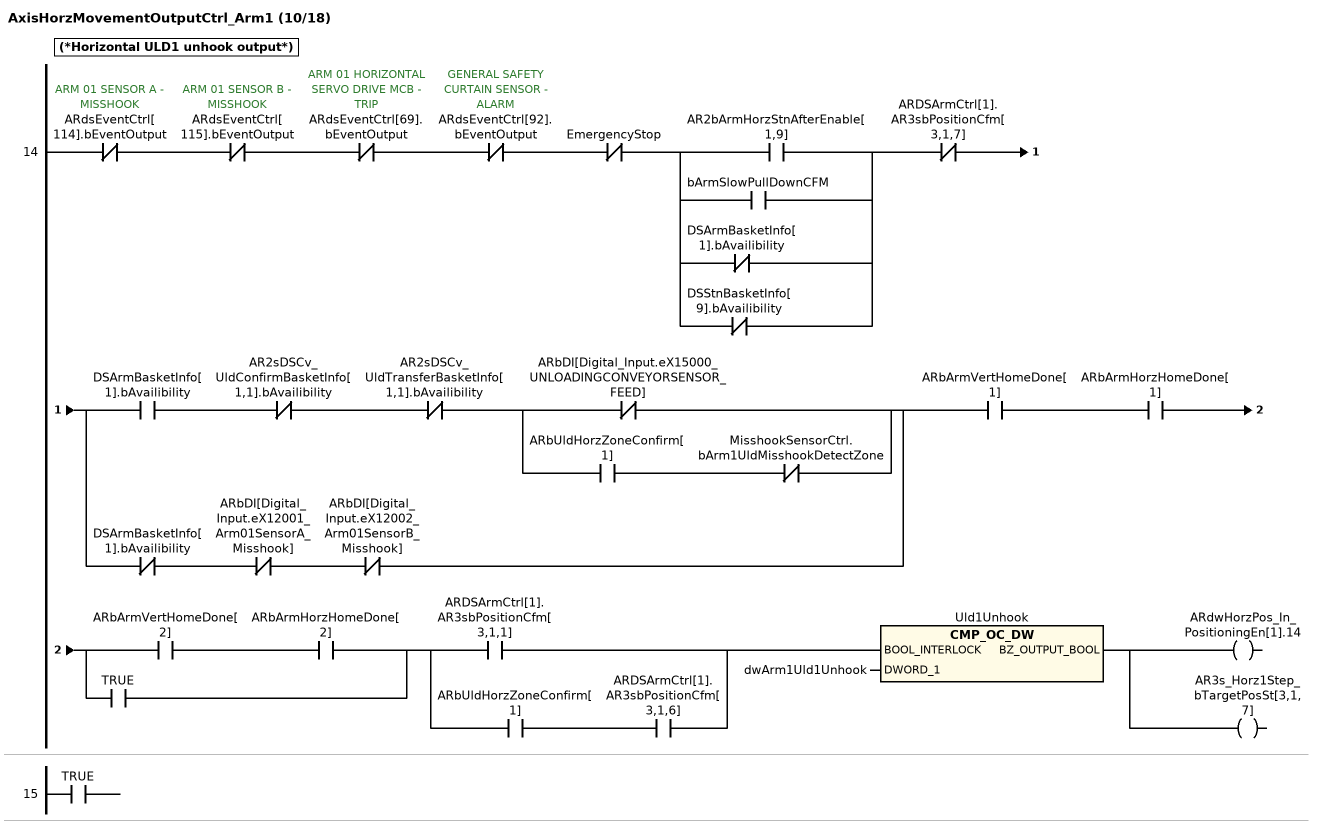
// NETWORK 14
//   ARdsEventCtrl[114].bEventOutput: ARM 01 SENSOR A - MISSHOOK
//   ARdsEventCtrl[115].bEventOutput: ARM 01 SENSOR B - MISSHOOK
//   ARdsEventCtrl[69].bEventOutput: ARM 01 HORIZONTAL SERVO DRIVE MCB - TRIP
//   ARdsEventCtrl[92].bEventOutput: GENERAL SAFETY CURTAIN SENSOR - ALARM
// label: (*Horizontal ULD1 unhook output*)
Uld1Unhook(BOOL_INTERLOCK := (((NOT ARdsEventCtrl[114].bEventOutput AND NOT ARdsEventCtrl[115].bEventOutput AND NOT ARdsEventCtrl[69].bEventOutput AND NOT ARdsEventCtrl[92].bEventOutput AND NOT EmergencyStop) AND (AR2bArmHorzStnAfterEnable[1,9] OR bArmSlowPullDownCFM OR NOT DSArmBasketInfo[1].bAvailibility OR NOT DSStnBasketInfo[9].bAvailibility)) AND NOT ARDSArmCtrl[1].AR3sbPositionCfm[3,1,7] AND (DSArmBasketInfo[1].bAvailibility AND NOT AR2sDSCv_UldConfirmBasketInfo[1,1].bAvailibility AND NOT AR2sDSCv_UldTransferBasketInfo[1,1].bAvailibility AND (NOT ARbDI[Digital_Input.eX15000_UNLOADINGCONVEYORSENSOR_FEED] OR ARbUldHorzZoneConfirm[1] AND NOT MisshookSensorCtrl.bArm1UldMisshookDetectZone) OR NOT DSArmBasketInfo[1].bAvailibility AND NOT ARbDI[Digital_Input.eX12001_Arm01SensorA_Misshook] AND NOT ARbDI[Digital_Input.eX12002_Arm01SensorB_Misshook])) AND ARbArmVertHomeDone[1] AND ARbArmHorzHomeDone[1] AND (ARbArmVertHomeDone[2] AND ARbArmHorzHomeDone[2] OR TRUE) AND (ARDSArmCtrl[1].AR3sbPositionCfm[3,1,1] OR ARbUldHorzZoneConfirm[1] AND ARDSArmCtrl[1].AR3sbPositionCfm[3,1,6]), DWORD_1 := dwArm1Uld1Unhook); // CMP_OC_DW
ARdwHorzPos_In_PositioningEn[1].14 := Uld1Unhook.BZ_OUTPUT_BOOL;
AR3s_Horz1Step_bTargetPosSt[3,1,7] := Uld1Unhook.BZ_OUTPUT_BOOL;

// NETWORK 15

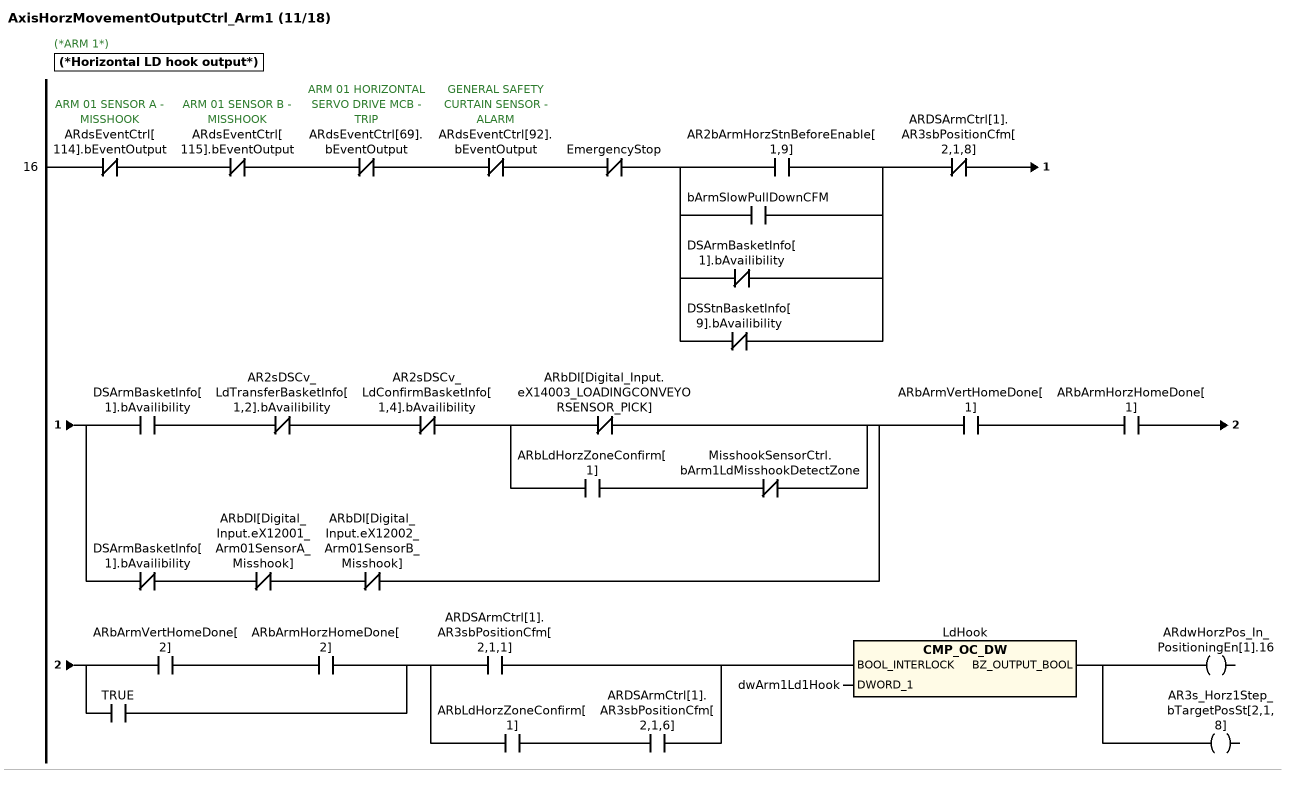
// NETWORK 16
// (*ARM 1*)
//   ARdsEventCtrl[114].bEventOutput: ARM 01 SENSOR A - MISSHOOK
//   ARdsEventCtrl[115].bEventOutput: ARM 01 SENSOR B - MISSHOOK
//   ARdsEventCtrl[69].bEventOutput: ARM 01 HORIZONTAL SERVO DRIVE MCB - TRIP
//   ARdsEventCtrl[92].bEventOutput: GENERAL SAFETY CURTAIN SENSOR - ALARM
// label: (*Horizontal LD hook output*)
LdHook(BOOL_INTERLOCK := (((NOT ARdsEventCtrl[114].bEventOutput AND NOT ARdsEventCtrl[115].bEventOutput AND NOT ARdsEventCtrl[69].bEventOutput AND NOT ARdsEventCtrl[92].bEventOutput AND NOT EmergencyStop) AND (AR2bArmHorzStnBeforeEnable[1,9] OR bArmSlowPullDownCFM OR NOT DSArmBasketInfo[1].bAvailibility OR NOT DSStnBasketInfo[9].bAvailibility)) AND NOT ARDSArmCtrl[1].AR3sbPositionCfm[2,1,8] AND (DSArmBasketInfo[1].bAvailibility AND NOT AR2sDSCv_LdTransferBasketInfo[1,2].bAvailibility AND NOT AR2sDSCv_LdConfirmBasketInfo[1,4].bAvailibility AND (NOT ARbDI[Digital_Input.eX14003_LOADINGCONVEYORSENSOR_PICK] OR ARbLdHorzZoneConfirm[1] AND NOT MisshookSensorCtrl.bArm1LdMisshookDetectZone) OR NOT DSArmBasketInfo[1].bAvailibility AND NOT ARbDI[Digital_Input.eX12001_Arm01SensorA_Misshook] AND NOT ARbDI[Digital_Input.eX12002_Arm01SensorB_Misshook])) AND ARbArmVertHomeDone[1] AND ARbArmHorzHomeDone[1] AND (ARbArmVertHomeDone[2] AND ARbArmHorzHomeDone[2] OR TRUE) AND (ARDSArmCtrl[1].AR3sbPositionCfm[2,1,1] OR ARbLdHorzZoneConfirm[1] AND ARDSArmCtrl[1].AR3sbPositionCfm[2,1,6]), DWORD_1 := dwArm1Ld1Hook); // CMP_OC_DW
ARdwHorzPos_In_PositioningEn[1].16 := LdHook.BZ_OUTPUT_BOOL;
AR3s_Horz1Step_bTargetPosSt[2,1,8] := LdHook.BZ_OUTPUT_BOOL;

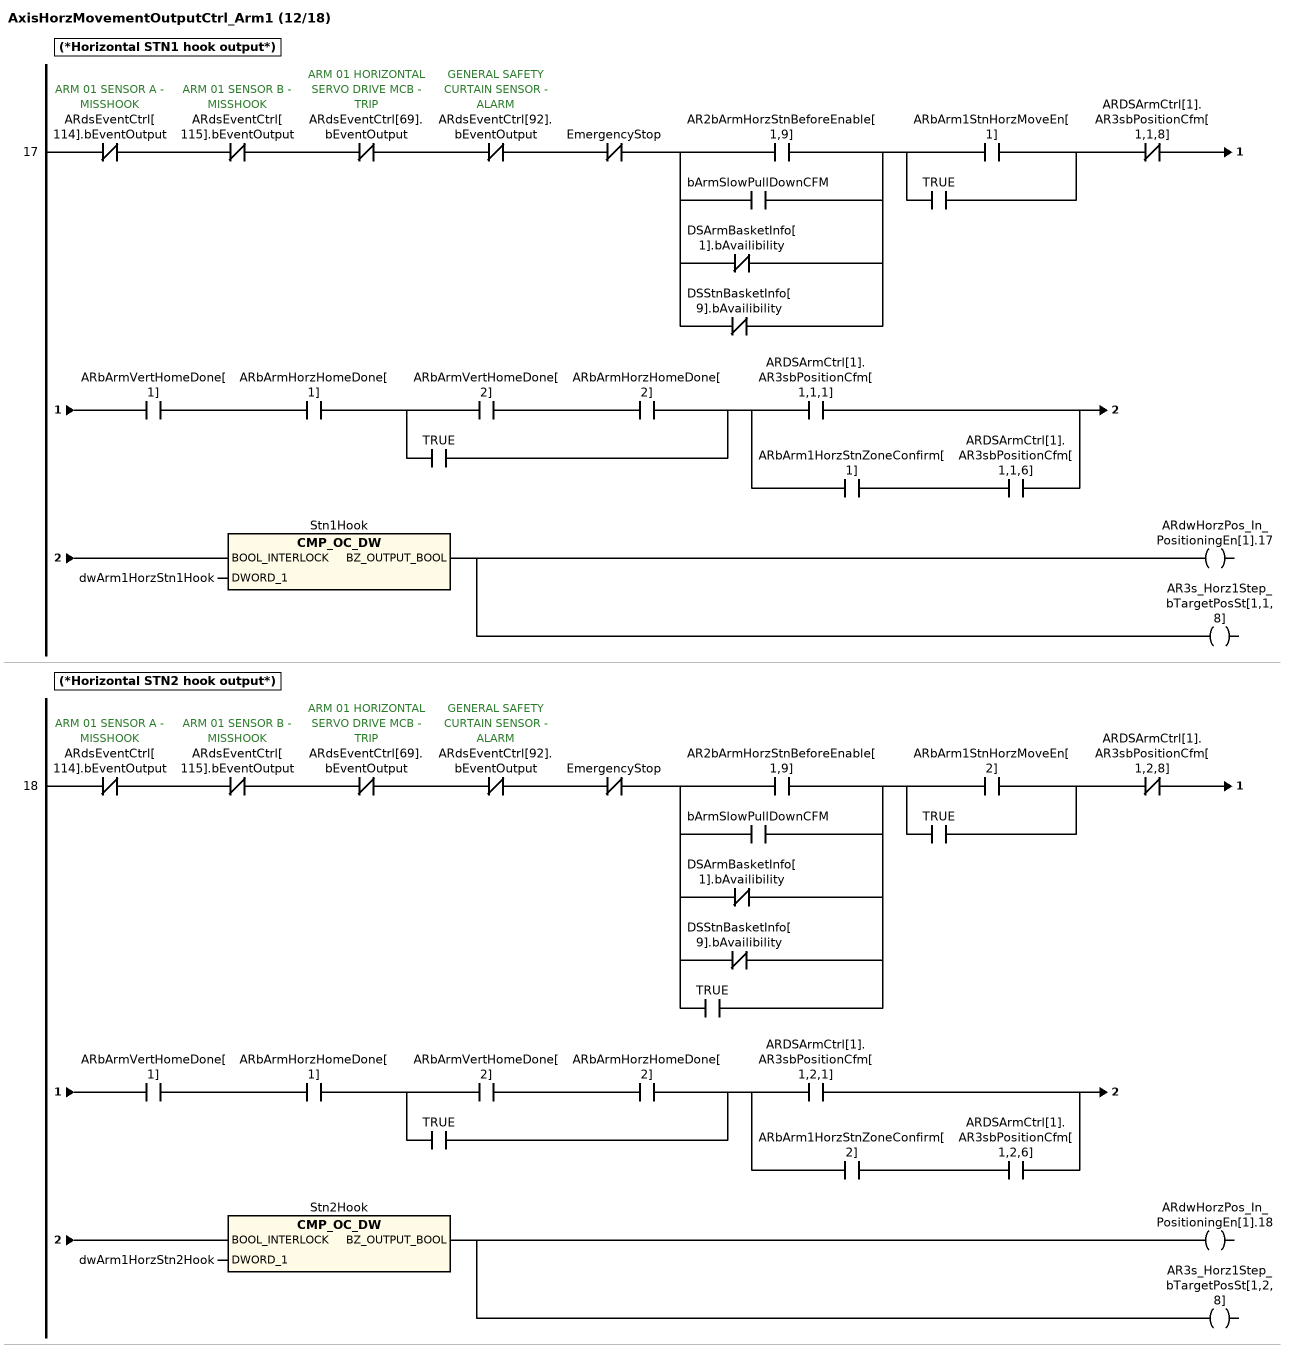
// NETWORK 17
//   ARdsEventCtrl[114].bEventOutput: ARM 01 SENSOR A - MISSHOOK
//   ARdsEventCtrl[115].bEventOutput: ARM 01 SENSOR B - MISSHOOK
//   ARdsEventCtrl[69].bEventOutput: ARM 01 HORIZONTAL SERVO DRIVE MCB - TRIP
//   ARdsEventCtrl[92].bEventOutput: GENERAL SAFETY CURTAIN SENSOR - ALARM
// label: (*Horizontal STN1 hook output*)
Stn1Hook(BOOL_INTERLOCK := ((NOT ARdsEventCtrl[114].bEventOutput AND NOT ARdsEventCtrl[115].bEventOutput AND NOT ARdsEventCtrl[69].bEventOutput AND NOT ARdsEventCtrl[92].bEventOutput AND NOT EmergencyStop) AND (AR2bArmHorzStnBeforeEnable[1,9] OR bArmSlowPullDownCFM OR NOT DSArmBasketInfo[1].bAvailibility OR NOT DSStnBasketInfo[9].bAvailibility) AND (ARbArm1StnHorzMoveEn[1] OR TRUE)) AND NOT ARDSArmCtrl[1].AR3sbPositionCfm[1,1,8] AND ARbArmVertHomeDone[1] AND ARbArmHorzHomeDone[1] AND (ARbArmVertHomeDone[2] AND ARbArmHorzHomeDone[2] OR TRUE) AND (ARDSArmCtrl[1].AR3sbPositionCfm[1,1,1] OR ARbArm1HorzStnZoneConfirm[1] AND ARDSArmCtrl[1].AR3sbPositionCfm[1,1,6]), DWORD_1 := dwArm1HorzStn1Hook); // CMP_OC_DW
ARdwHorzPos_In_PositioningEn[1].17 := Stn1Hook.BZ_OUTPUT_BOOL;
AR3s_Horz1Step_bTargetPosSt[1,1,8] := Stn1Hook.BZ_OUTPUT_BOOL;

// NETWORK 18
//   ARdsEventCtrl[114].bEventOutput: ARM 01 SENSOR A - MISSHOOK
//   ARdsEventCtrl[115].bEventOutput: ARM 01 SENSOR B - MISSHOOK
//   ARdsEventCtrl[69].bEventOutput: ARM 01 HORIZONTAL SERVO DRIVE MCB - TRIP
//   ARdsEventCtrl[92].bEventOutput: GENERAL SAFETY CURTAIN SENSOR - ALARM
// label: (*Horizontal STN2 hook output*)
Stn2Hook(BOOL_INTERLOCK := ((NOT ARdsEventCtrl[114].bEventOutput AND NOT ARdsEventCtrl[115].bEventOutput AND NOT ARdsEventCtrl[69].bEventOutput AND NOT ARdsEventCtrl[92].bEventOutput AND NOT EmergencyStop) AND (AR2bArmHorzStnBeforeEnable[1,9] OR bArmSlowPullDownCFM OR NOT DSArmBasketInfo[1].bAvailibility OR NOT DSStnBasketInfo[9].bAvailibility OR TRUE) AND (ARbArm1StnHorzMoveEn[2] OR TRUE)) AND NOT ARDSArmCtrl[1].AR3sbPositionCfm[1,2,8] AND ARbArmVertHomeDone[1] AND ARbArmHorzHomeDone[1] AND (ARbArmVertHomeDone[2] AND ARbArmHorzHomeDone[2] OR TRUE) AND (ARDSArmCtrl[1].AR3sbPositionCfm[1,2,1] OR ARbArm1HorzStnZoneConfirm[2] AND ARDSArmCtrl[1].AR3sbPositionCfm[1,2,6]), DWORD_1 := dwArm1HorzStn2Hook); // CMP_OC_DW
ARdwHorzPos_In_PositioningEn[1].18 := Stn2Hook.BZ_OUTPUT_BOOL;
AR3s_Horz1Step_bTargetPosSt[1,2,8] := Stn2Hook.BZ_OUTPUT_BOOL;

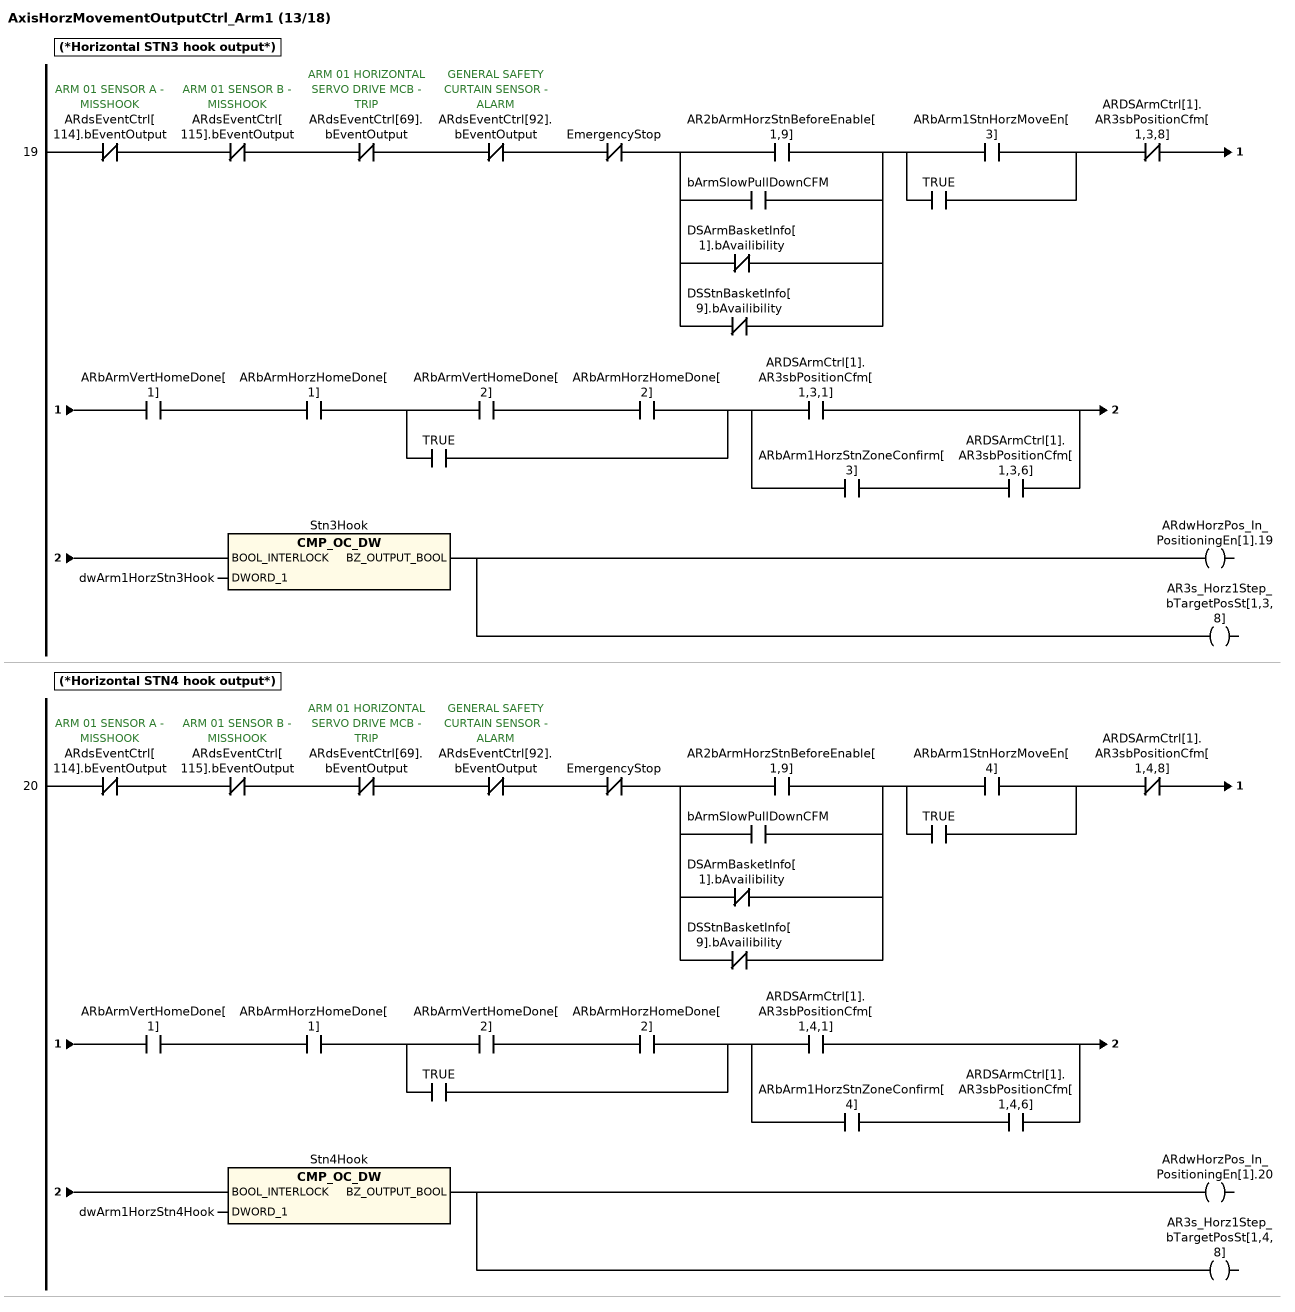
// NETWORK 19
//   ARdsEventCtrl[114].bEventOutput: ARM 01 SENSOR A - MISSHOOK
//   ARdsEventCtrl[115].bEventOutput: ARM 01 SENSOR B - MISSHOOK
//   ARdsEventCtrl[69].bEventOutput: ARM 01 HORIZONTAL SERVO DRIVE MCB - TRIP
//   ARdsEventCtrl[92].bEventOutput: GENERAL SAFETY CURTAIN SENSOR - ALARM
// label: (*Horizontal STN3 hook output*)
Stn3Hook(BOOL_INTERLOCK := ((NOT ARdsEventCtrl[114].bEventOutput AND NOT ARdsEventCtrl[115].bEventOutput AND NOT ARdsEventCtrl[69].bEventOutput AND NOT ARdsEventCtrl[92].bEventOutput AND NOT EmergencyStop) AND (AR2bArmHorzStnBeforeEnable[1,9] OR bArmSlowPullDownCFM OR NOT DSArmBasketInfo[1].bAvailibility OR NOT DSStnBasketInfo[9].bAvailibility) AND (ARbArm1StnHorzMoveEn[3] OR TRUE)) AND NOT ARDSArmCtrl[1].AR3sbPositionCfm[1,3,8] AND ARbArmVertHomeDone[1] AND ARbArmHorzHomeDone[1] AND (ARbArmVertHomeDone[2] AND ARbArmHorzHomeDone[2] OR TRUE) AND (ARDSArmCtrl[1].AR3sbPositionCfm[1,3,1] OR ARbArm1HorzStnZoneConfirm[3] AND ARDSArmCtrl[1].AR3sbPositionCfm[1,3,6]), DWORD_1 := dwArm1HorzStn3Hook); // CMP_OC_DW
ARdwHorzPos_In_PositioningEn[1].19 := Stn3Hook.BZ_OUTPUT_BOOL;
AR3s_Horz1Step_bTargetPosSt[1,3,8] := Stn3Hook.BZ_OUTPUT_BOOL;

// NETWORK 20
//   ARdsEventCtrl[114].bEventOutput: ARM 01 SENSOR A - MISSHOOK
//   ARdsEventCtrl[115].bEventOutput: ARM 01 SENSOR B - MISSHOOK
//   ARdsEventCtrl[69].bEventOutput: ARM 01 HORIZONTAL SERVO DRIVE MCB - TRIP
//   ARdsEventCtrl[92].bEventOutput: GENERAL SAFETY CURTAIN SENSOR - ALARM
// label: (*Horizontal STN4 hook output*)
Stn4Hook(BOOL_INTERLOCK := ((NOT ARdsEventCtrl[114].bEventOutput AND NOT ARdsEventCtrl[115].bEventOutput AND NOT ARdsEventCtrl[69].bEventOutput AND NOT ARdsEventCtrl[92].bEventOutput AND NOT EmergencyStop) AND (AR2bArmHorzStnBeforeEnable[1,9] OR bArmSlowPullDownCFM OR NOT DSArmBasketInfo[1].bAvailibility OR NOT DSStnBasketInfo[9].bAvailibility) AND (ARbArm1StnHorzMoveEn[4] OR TRUE)) AND NOT ARDSArmCtrl[1].AR3sbPositionCfm[1,4,8] AND ARbArmVertHomeDone[1] AND ARbArmHorzHomeDone[1] AND (ARbArmVertHomeDone[2] AND ARbArmHorzHomeDone[2] OR TRUE) AND (ARDSArmCtrl[1].AR3sbPositionCfm[1,4,1] OR ARbArm1HorzStnZoneConfirm[4] AND ARDSArmCtrl[1].AR3sbPositionCfm[1,4,6]), DWORD_1 := dwArm1HorzStn4Hook); // CMP_OC_DW
ARdwHorzPos_In_PositioningEn[1].20 := Stn4Hook.BZ_OUTPUT_BOOL;
AR3s_Horz1Step_bTargetPosSt[1,4,8] := Stn4Hook.BZ_OUTPUT_BOOL;

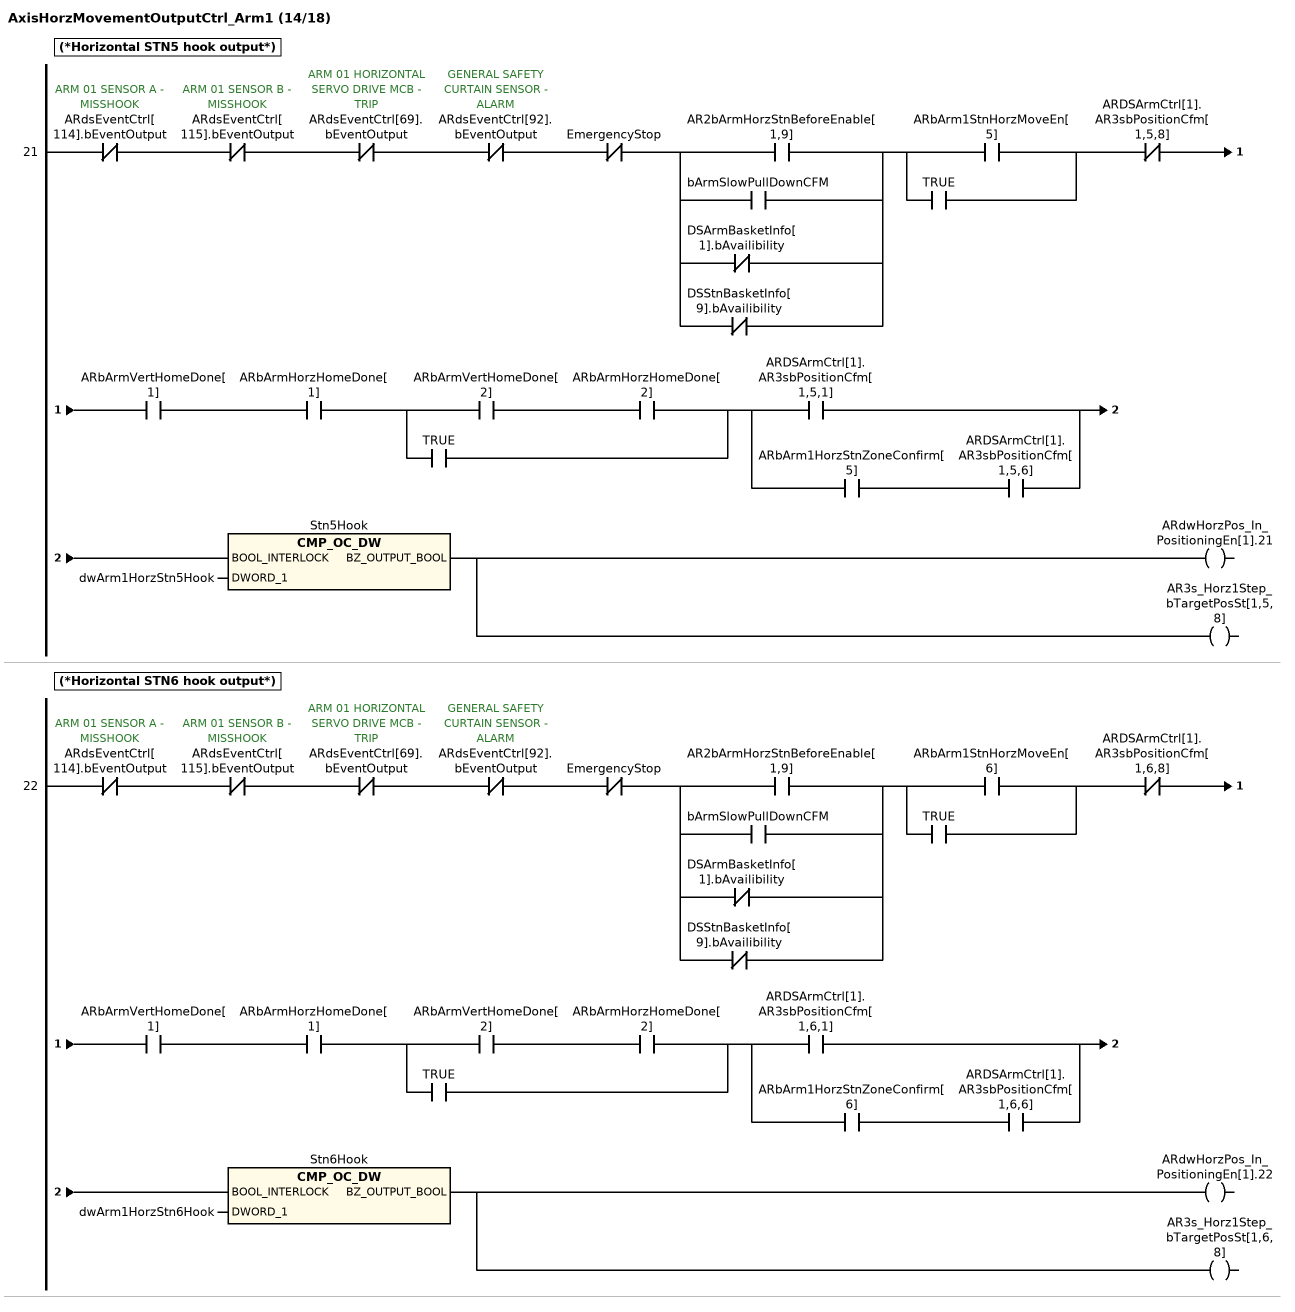
// NETWORK 21
//   ARdsEventCtrl[114].bEventOutput: ARM 01 SENSOR A - MISSHOOK
//   ARdsEventCtrl[115].bEventOutput: ARM 01 SENSOR B - MISSHOOK
//   ARdsEventCtrl[69].bEventOutput: ARM 01 HORIZONTAL SERVO DRIVE MCB - TRIP
//   ARdsEventCtrl[92].bEventOutput: GENERAL SAFETY CURTAIN SENSOR - ALARM
// label: (*Horizontal STN5 hook output*)
Stn5Hook(BOOL_INTERLOCK := ((NOT ARdsEventCtrl[114].bEventOutput AND NOT ARdsEventCtrl[115].bEventOutput AND NOT ARdsEventCtrl[69].bEventOutput AND NOT ARdsEventCtrl[92].bEventOutput AND NOT EmergencyStop) AND (AR2bArmHorzStnBeforeEnable[1,9] OR bArmSlowPullDownCFM OR NOT DSArmBasketInfo[1].bAvailibility OR NOT DSStnBasketInfo[9].bAvailibility) AND (ARbArm1StnHorzMoveEn[5] OR TRUE)) AND NOT ARDSArmCtrl[1].AR3sbPositionCfm[1,5,8] AND ARbArmVertHomeDone[1] AND ARbArmHorzHomeDone[1] AND (ARbArmVertHomeDone[2] AND ARbArmHorzHomeDone[2] OR TRUE) AND (ARDSArmCtrl[1].AR3sbPositionCfm[1,5,1] OR ARbArm1HorzStnZoneConfirm[5] AND ARDSArmCtrl[1].AR3sbPositionCfm[1,5,6]), DWORD_1 := dwArm1HorzStn5Hook); // CMP_OC_DW
ARdwHorzPos_In_PositioningEn[1].21 := Stn5Hook.BZ_OUTPUT_BOOL;
AR3s_Horz1Step_bTargetPosSt[1,5,8] := Stn5Hook.BZ_OUTPUT_BOOL;

// NETWORK 22
//   ARdsEventCtrl[114].bEventOutput: ARM 01 SENSOR A - MISSHOOK
//   ARdsEventCtrl[115].bEventOutput: ARM 01 SENSOR B - MISSHOOK
//   ARdsEventCtrl[69].bEventOutput: ARM 01 HORIZONTAL SERVO DRIVE MCB - TRIP
//   ARdsEventCtrl[92].bEventOutput: GENERAL SAFETY CURTAIN SENSOR - ALARM
// label: (*Horizontal STN6 hook output*)
Stn6Hook(BOOL_INTERLOCK := ((NOT ARdsEventCtrl[114].bEventOutput AND NOT ARdsEventCtrl[115].bEventOutput AND NOT ARdsEventCtrl[69].bEventOutput AND NOT ARdsEventCtrl[92].bEventOutput AND NOT EmergencyStop) AND ((AR2bArmHorzStnBeforeEnable[1,9] OR bArmSlowPullDownCFM OR NOT DSArmBasketInfo[1].bAvailibility OR NOT DSStnBasketInfo[9].bAvailibility) AND (ARbArm1StnHorzMoveEn[6] OR TRUE))) AND NOT ARDSArmCtrl[1].AR3sbPositionCfm[1,6,8] AND ARbArmVertHomeDone[1] AND ARbArmHorzHomeDone[1] AND (ARbArmVertHomeDone[2] AND ARbArmHorzHomeDone[2] OR TRUE) AND (ARDSArmCtrl[1].AR3sbPositionCfm[1,6,1] OR ARbArm1HorzStnZoneConfirm[6] AND ARDSArmCtrl[1].AR3sbPositionCfm[1,6,6]), DWORD_1 := dwArm1HorzStn6Hook); // CMP_OC_DW
ARdwHorzPos_In_PositioningEn[1].22 := Stn6Hook.BZ_OUTPUT_BOOL;
AR3s_Horz1Step_bTargetPosSt[1,6,8] := Stn6Hook.BZ_OUTPUT_BOOL;

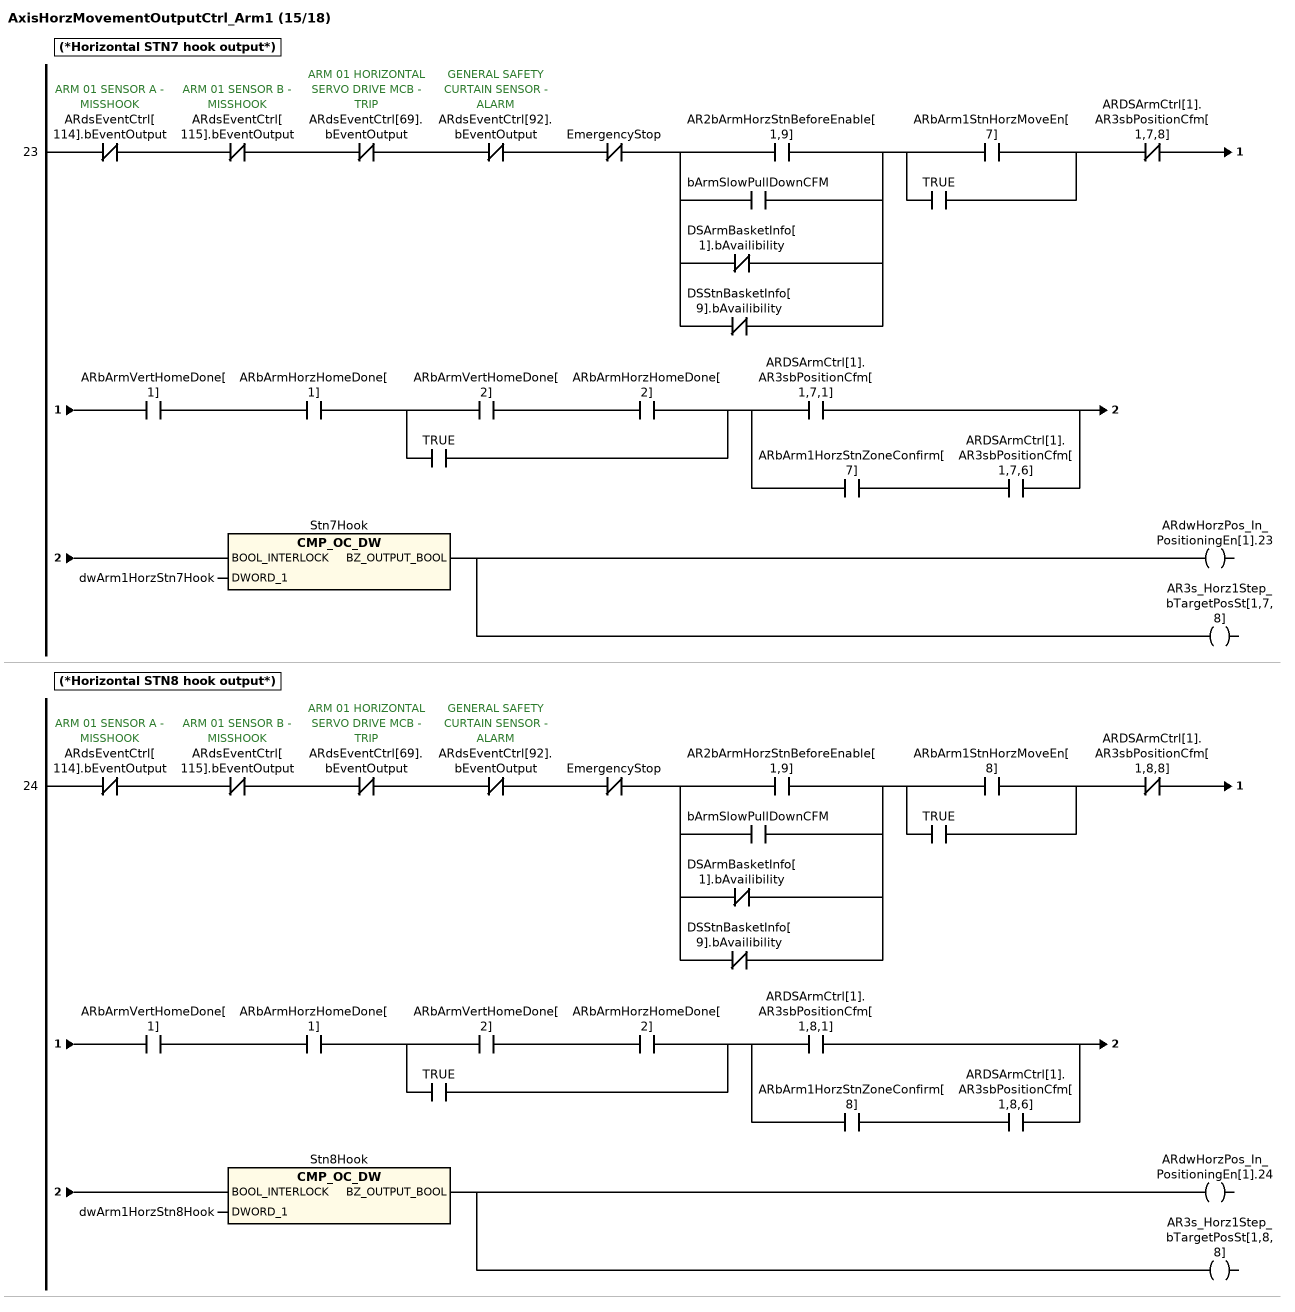
// NETWORK 23
//   ARdsEventCtrl[114].bEventOutput: ARM 01 SENSOR A - MISSHOOK
//   ARdsEventCtrl[115].bEventOutput: ARM 01 SENSOR B - MISSHOOK
//   ARdsEventCtrl[69].bEventOutput: ARM 01 HORIZONTAL SERVO DRIVE MCB - TRIP
//   ARdsEventCtrl[92].bEventOutput: GENERAL SAFETY CURTAIN SENSOR - ALARM
// label: (*Horizontal STN7 hook output*)
Stn7Hook(BOOL_INTERLOCK := ((NOT ARdsEventCtrl[114].bEventOutput AND NOT ARdsEventCtrl[115].bEventOutput AND NOT ARdsEventCtrl[69].bEventOutput AND NOT ARdsEventCtrl[92].bEventOutput AND NOT EmergencyStop) AND (AR2bArmHorzStnBeforeEnable[1,9] OR bArmSlowPullDownCFM OR NOT DSArmBasketInfo[1].bAvailibility OR NOT DSStnBasketInfo[9].bAvailibility) AND (ARbArm1StnHorzMoveEn[7] OR TRUE)) AND NOT ARDSArmCtrl[1].AR3sbPositionCfm[1,7,8] AND ARbArmVertHomeDone[1] AND ARbArmHorzHomeDone[1] AND (ARbArmVertHomeDone[2] AND ARbArmHorzHomeDone[2] OR TRUE) AND (ARDSArmCtrl[1].AR3sbPositionCfm[1,7,1] OR ARbArm1HorzStnZoneConfirm[7] AND ARDSArmCtrl[1].AR3sbPositionCfm[1,7,6]), DWORD_1 := dwArm1HorzStn7Hook); // CMP_OC_DW
ARdwHorzPos_In_PositioningEn[1].23 := Stn7Hook.BZ_OUTPUT_BOOL;
AR3s_Horz1Step_bTargetPosSt[1,7,8] := Stn7Hook.BZ_OUTPUT_BOOL;

// NETWORK 24
//   ARdsEventCtrl[114].bEventOutput: ARM 01 SENSOR A - MISSHOOK
//   ARdsEventCtrl[115].bEventOutput: ARM 01 SENSOR B - MISSHOOK
//   ARdsEventCtrl[69].bEventOutput: ARM 01 HORIZONTAL SERVO DRIVE MCB - TRIP
//   ARdsEventCtrl[92].bEventOutput: GENERAL SAFETY CURTAIN SENSOR - ALARM
// label: (*Horizontal STN8 hook output*)
Stn8Hook(BOOL_INTERLOCK := (NOT ARdsEventCtrl[114].bEventOutput AND NOT ARdsEventCtrl[115].bEventOutput AND NOT ARdsEventCtrl[69].bEventOutput AND NOT ARdsEventCtrl[92].bEventOutput AND NOT EmergencyStop AND (AR2bArmHorzStnBeforeEnable[1,9] OR bArmSlowPullDownCFM OR NOT DSArmBasketInfo[1].bAvailibility OR NOT DSStnBasketInfo[9].bAvailibility) AND (ARbArm1StnHorzMoveEn[8] OR TRUE)) AND NOT ARDSArmCtrl[1].AR3sbPositionCfm[1,8,8] AND ARbArmVertHomeDone[1] AND ARbArmHorzHomeDone[1] AND (ARbArmVertHomeDone[2] AND ARbArmHorzHomeDone[2] OR TRUE) AND (ARDSArmCtrl[1].AR3sbPositionCfm[1,8,1] OR ARbArm1HorzStnZoneConfirm[8] AND ARDSArmCtrl[1].AR3sbPositionCfm[1,8,6]), DWORD_1 := dwArm1HorzStn8Hook); // CMP_OC_DW
ARdwHorzPos_In_PositioningEn[1].24 := Stn8Hook.BZ_OUTPUT_BOOL;
AR3s_Horz1Step_bTargetPosSt[1,8,8] := Stn8Hook.BZ_OUTPUT_BOOL;

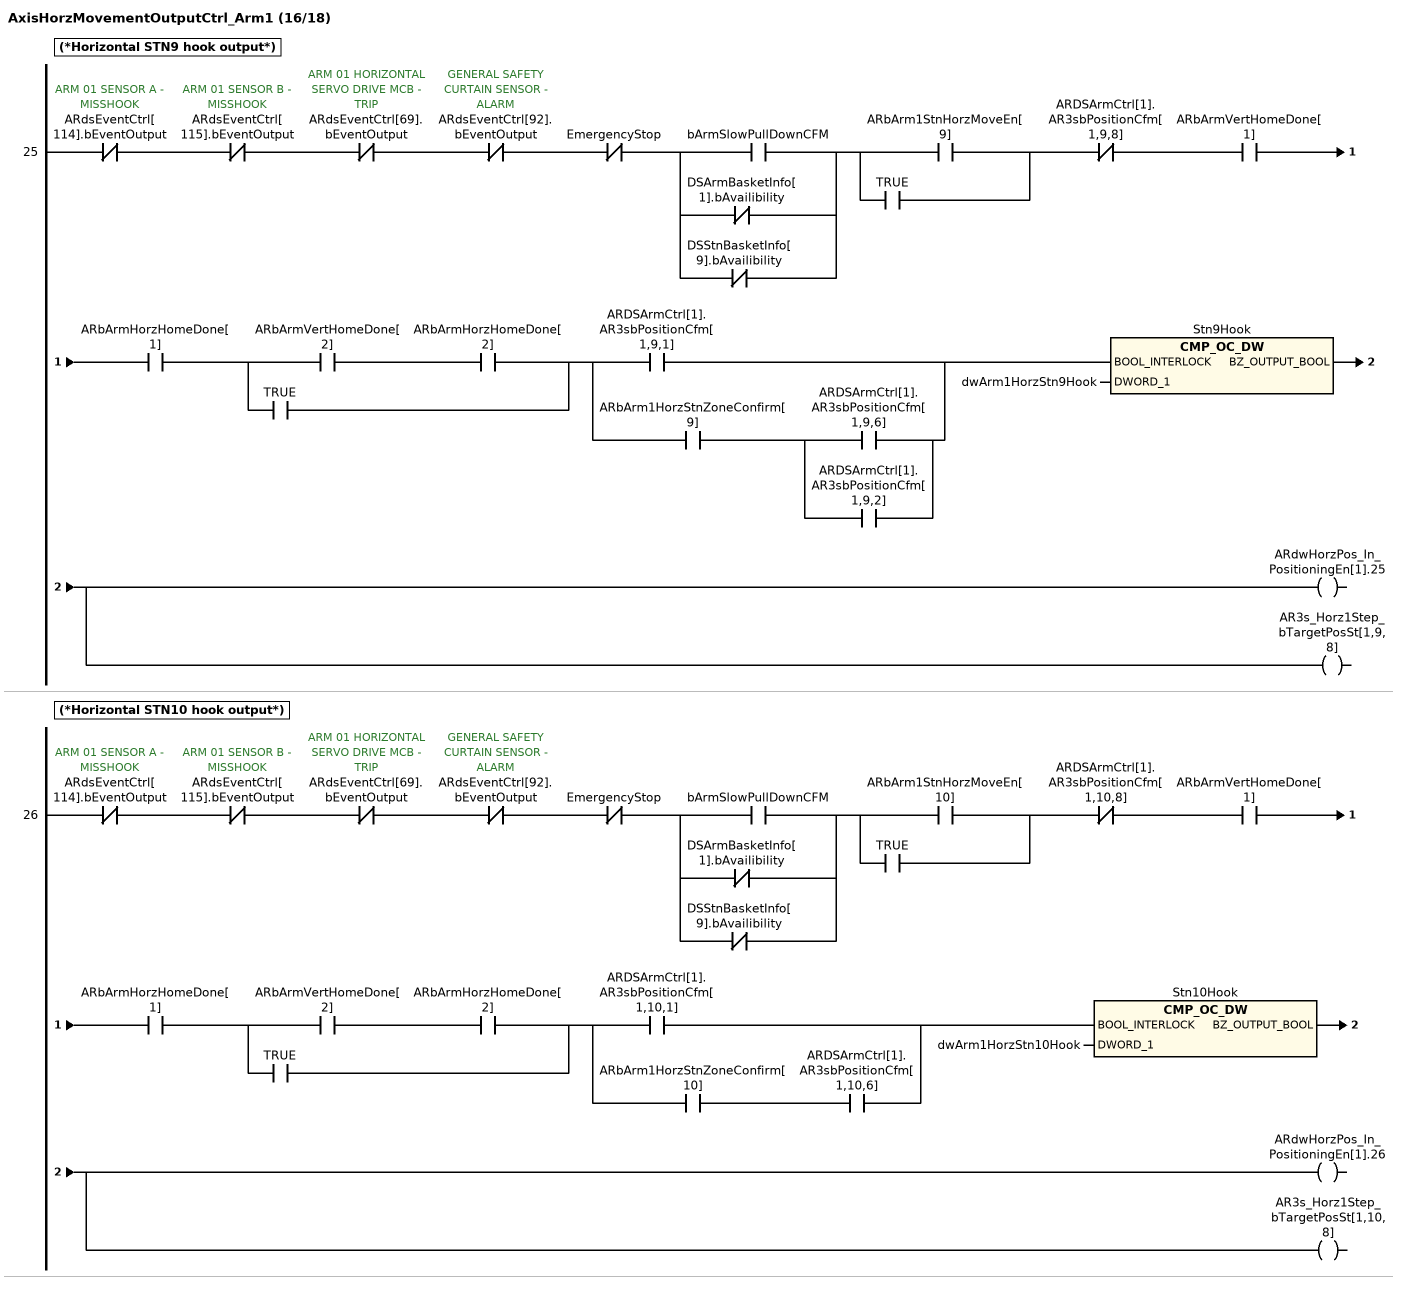
// NETWORK 25
//   ARdsEventCtrl[114].bEventOutput: ARM 01 SENSOR A - MISSHOOK
//   ARdsEventCtrl[115].bEventOutput: ARM 01 SENSOR B - MISSHOOK
//   ARdsEventCtrl[69].bEventOutput: ARM 01 HORIZONTAL SERVO DRIVE MCB - TRIP
//   ARdsEventCtrl[92].bEventOutput: GENERAL SAFETY CURTAIN SENSOR - ALARM
// label: (*Horizontal STN9 hook output*)
Stn9Hook(BOOL_INTERLOCK := ((NOT ARdsEventCtrl[114].bEventOutput AND NOT ARdsEventCtrl[115].bEventOutput AND NOT ARdsEventCtrl[69].bEventOutput AND NOT ARdsEventCtrl[92].bEventOutput AND NOT EmergencyStop) AND (bArmSlowPullDownCFM OR NOT DSArmBasketInfo[1].bAvailibility OR NOT DSStnBasketInfo[9].bAvailibility) AND (ARbArm1StnHorzMoveEn[9] OR TRUE)) AND NOT ARDSArmCtrl[1].AR3sbPositionCfm[1,9,8] AND ARbArmVertHomeDone[1] AND ARbArmHorzHomeDone[1] AND (ARbArmVertHomeDone[2] AND ARbArmHorzHomeDone[2] OR TRUE) AND (ARDSArmCtrl[1].AR3sbPositionCfm[1,9,1] OR ARbArm1HorzStnZoneConfirm[9] AND (ARDSArmCtrl[1].AR3sbPositionCfm[1,9,6] OR ARDSArmCtrl[1].AR3sbPositionCfm[1,9,2])), DWORD_1 := dwArm1HorzStn9Hook); // CMP_OC_DW
ARdwHorzPos_In_PositioningEn[1].25 := Stn9Hook.BZ_OUTPUT_BOOL;
AR3s_Horz1Step_bTargetPosSt[1,9,8] := Stn9Hook.BZ_OUTPUT_BOOL;

// NETWORK 26
//   ARdsEventCtrl[114].bEventOutput: ARM 01 SENSOR A - MISSHOOK
//   ARdsEventCtrl[115].bEventOutput: ARM 01 SENSOR B - MISSHOOK
//   ARdsEventCtrl[69].bEventOutput: ARM 01 HORIZONTAL SERVO DRIVE MCB - TRIP
//   ARdsEventCtrl[92].bEventOutput: GENERAL SAFETY CURTAIN SENSOR - ALARM
// label: (*Horizontal STN10 hook output*)
Stn10Hook(BOOL_INTERLOCK := ((NOT ARdsEventCtrl[114].bEventOutput AND NOT ARdsEventCtrl[115].bEventOutput AND NOT ARdsEventCtrl[69].bEventOutput AND NOT ARdsEventCtrl[92].bEventOutput AND NOT EmergencyStop) AND (bArmSlowPullDownCFM OR NOT DSArmBasketInfo[1].bAvailibility OR NOT DSStnBasketInfo[9].bAvailibility) AND (ARbArm1StnHorzMoveEn[10] OR TRUE)) AND NOT ARDSArmCtrl[1].AR3sbPositionCfm[1,10,8] AND ARbArmVertHomeDone[1] AND ARbArmHorzHomeDone[1] AND (ARbArmVertHomeDone[2] AND ARbArmHorzHomeDone[2] OR TRUE) AND (ARDSArmCtrl[1].AR3sbPositionCfm[1,10,1] OR ARbArm1HorzStnZoneConfirm[10] AND ARDSArmCtrl[1].AR3sbPositionCfm[1,10,6]), DWORD_1 := dwArm1HorzStn10Hook); // CMP_OC_DW
ARdwHorzPos_In_PositioningEn[1].26 := Stn10Hook.BZ_OUTPUT_BOOL;
AR3s_Horz1Step_bTargetPosSt[1,10,8] := Stn10Hook.BZ_OUTPUT_BOOL;

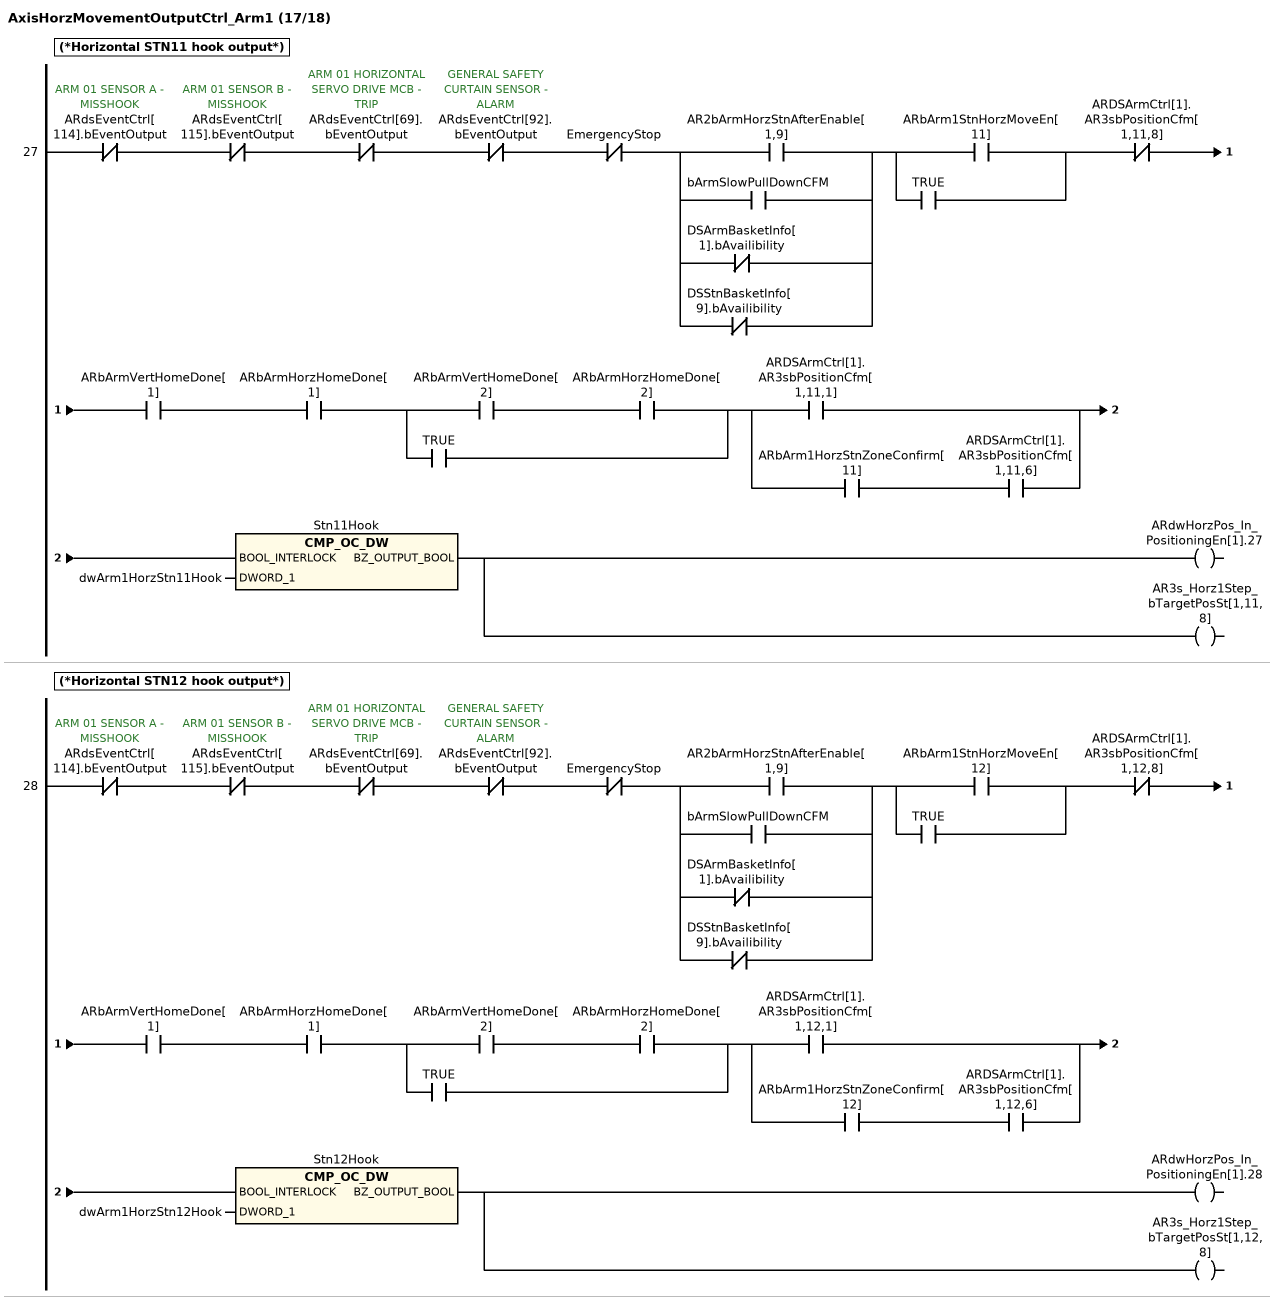
// NETWORK 27
//   ARdsEventCtrl[114].bEventOutput: ARM 01 SENSOR A - MISSHOOK
//   ARdsEventCtrl[115].bEventOutput: ARM 01 SENSOR B - MISSHOOK
//   ARdsEventCtrl[69].bEventOutput: ARM 01 HORIZONTAL SERVO DRIVE MCB - TRIP
//   ARdsEventCtrl[92].bEventOutput: GENERAL SAFETY CURTAIN SENSOR - ALARM
// label: (*Horizontal STN11 hook output*)
Stn11Hook(BOOL_INTERLOCK := ((NOT ARdsEventCtrl[114].bEventOutput AND NOT ARdsEventCtrl[115].bEventOutput AND NOT ARdsEventCtrl[69].bEventOutput AND NOT ARdsEventCtrl[92].bEventOutput AND NOT EmergencyStop) AND (AR2bArmHorzStnAfterEnable[1,9] OR bArmSlowPullDownCFM OR NOT DSArmBasketInfo[1].bAvailibility OR NOT DSStnBasketInfo[9].bAvailibility) AND (ARbArm1StnHorzMoveEn[11] OR TRUE)) AND NOT ARDSArmCtrl[1].AR3sbPositionCfm[1,11,8] AND ARbArmVertHomeDone[1] AND ARbArmHorzHomeDone[1] AND (ARbArmVertHomeDone[2] AND ARbArmHorzHomeDone[2] OR TRUE) AND (ARDSArmCtrl[1].AR3sbPositionCfm[1,11,1] OR ARbArm1HorzStnZoneConfirm[11] AND ARDSArmCtrl[1].AR3sbPositionCfm[1,11,6]), DWORD_1 := dwArm1HorzStn11Hook); // CMP_OC_DW
ARdwHorzPos_In_PositioningEn[1].27 := Stn11Hook.BZ_OUTPUT_BOOL;
AR3s_Horz1Step_bTargetPosSt[1,11,8] := Stn11Hook.BZ_OUTPUT_BOOL;

// NETWORK 28
//   ARdsEventCtrl[114].bEventOutput: ARM 01 SENSOR A - MISSHOOK
//   ARdsEventCtrl[115].bEventOutput: ARM 01 SENSOR B - MISSHOOK
//   ARdsEventCtrl[69].bEventOutput: ARM 01 HORIZONTAL SERVO DRIVE MCB - TRIP
//   ARdsEventCtrl[92].bEventOutput: GENERAL SAFETY CURTAIN SENSOR - ALARM
// label: (*Horizontal STN12 hook output*)
Stn12Hook(BOOL_INTERLOCK := ((NOT ARdsEventCtrl[114].bEventOutput AND NOT ARdsEventCtrl[115].bEventOutput AND NOT ARdsEventCtrl[69].bEventOutput AND NOT ARdsEventCtrl[92].bEventOutput AND NOT EmergencyStop) AND (AR2bArmHorzStnAfterEnable[1,9] OR bArmSlowPullDownCFM OR NOT DSArmBasketInfo[1].bAvailibility OR NOT DSStnBasketInfo[9].bAvailibility) AND (ARbArm1StnHorzMoveEn[12] OR TRUE)) AND NOT ARDSArmCtrl[1].AR3sbPositionCfm[1,12,8] AND ARbArmVertHomeDone[1] AND ARbArmHorzHomeDone[1] AND (ARbArmVertHomeDone[2] AND ARbArmHorzHomeDone[2] OR TRUE) AND (ARDSArmCtrl[1].AR3sbPositionCfm[1,12,1] OR ARbArm1HorzStnZoneConfirm[12] AND ARDSArmCtrl[1].AR3sbPositionCfm[1,12,6]), DWORD_1 := dwArm1HorzStn12Hook); // CMP_OC_DW
ARdwHorzPos_In_PositioningEn[1].28 := Stn12Hook.BZ_OUTPUT_BOOL;
AR3s_Horz1Step_bTargetPosSt[1,12,8] := Stn12Hook.BZ_OUTPUT_BOOL;

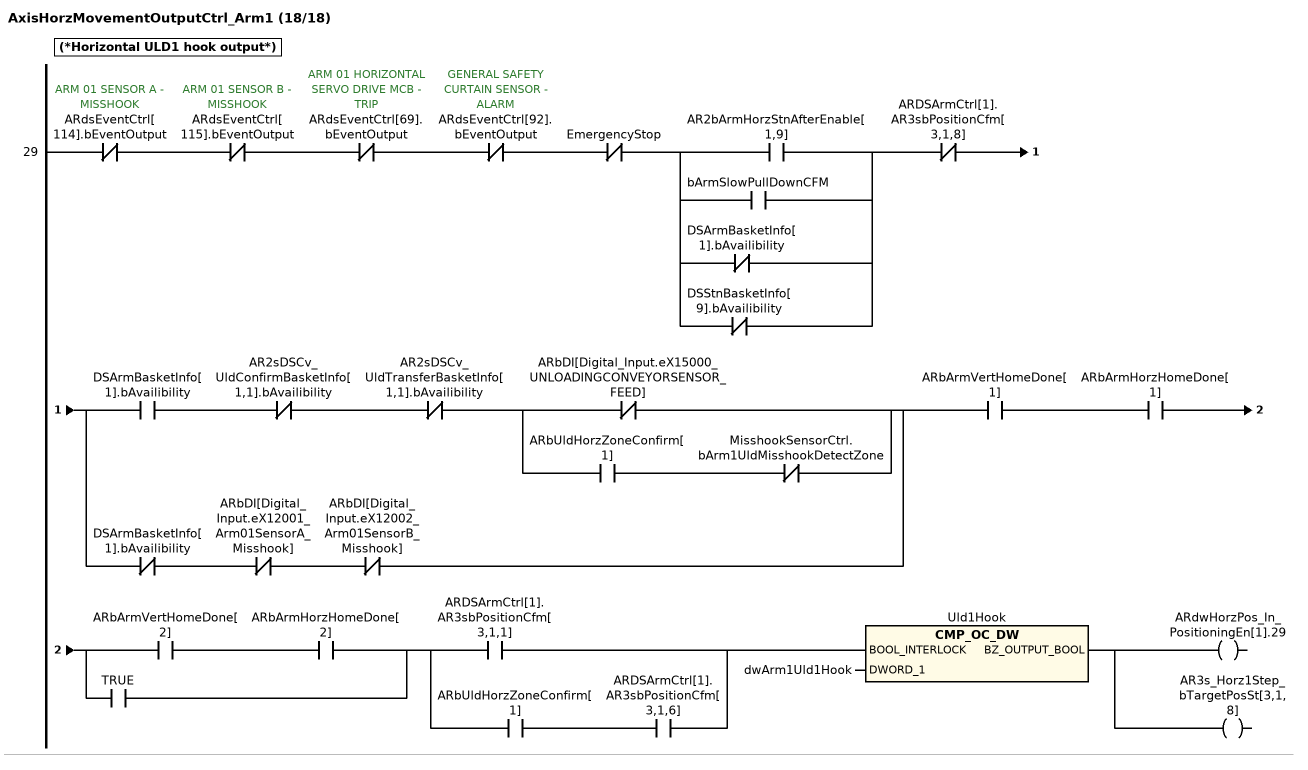
// NETWORK 29
//   ARdsEventCtrl[114].bEventOutput: ARM 01 SENSOR A - MISSHOOK
//   ARdsEventCtrl[115].bEventOutput: ARM 01 SENSOR B - MISSHOOK
//   ARdsEventCtrl[69].bEventOutput: ARM 01 HORIZONTAL SERVO DRIVE MCB - TRIP
//   ARdsEventCtrl[92].bEventOutput: GENERAL SAFETY CURTAIN SENSOR - ALARM
// label: (*Horizontal ULD1 hook output*)
Uld1Hook(BOOL_INTERLOCK := (((NOT ARdsEventCtrl[114].bEventOutput AND NOT ARdsEventCtrl[115].bEventOutput AND NOT ARdsEventCtrl[69].bEventOutput AND NOT ARdsEventCtrl[92].bEventOutput AND NOT EmergencyStop) AND (AR2bArmHorzStnAfterEnable[1,9] OR bArmSlowPullDownCFM OR NOT DSArmBasketInfo[1].bAvailibility OR NOT DSStnBasketInfo[9].bAvailibility)) AND NOT ARDSArmCtrl[1].AR3sbPositionCfm[3,1,8] AND (DSArmBasketInfo[1].bAvailibility AND NOT AR2sDSCv_UldConfirmBasketInfo[1,1].bAvailibility AND NOT AR2sDSCv_UldTransferBasketInfo[1,1].bAvailibility AND (NOT ARbDI[Digital_Input.eX15000_UNLOADINGCONVEYORSENSOR_FEED] OR ARbUldHorzZoneConfirm[1] AND NOT MisshookSensorCtrl.bArm1UldMisshookDetectZone) OR NOT DSArmBasketInfo[1].bAvailibility AND NOT ARbDI[Digital_Input.eX12001_Arm01SensorA_Misshook] AND NOT ARbDI[Digital_Input.eX12002_Arm01SensorB_Misshook])) AND ARbArmVertHomeDone[1] AND ARbArmHorzHomeDone[1] AND (ARbArmVertHomeDone[2] AND ARbArmHorzHomeDone[2] OR TRUE) AND (ARDSArmCtrl[1].AR3sbPositionCfm[3,1,1] OR ARbUldHorzZoneConfirm[1] AND ARDSArmCtrl[1].AR3sbPositionCfm[3,1,6]), DWORD_1 := dwArm1Uld1Hook); // CMP_OC_DW
ARdwHorzPos_In_PositioningEn[1].29 := Uld1Hook.BZ_OUTPUT_BOOL;
AR3s_Horz1Step_bTargetPosSt[3,1,8] := Uld1Hook.BZ_OUTPUT_BOOL;

END_PROGRAM

// ---- FBs/B_JKS_OldFB/Word to Bit/CMP_OC_DW.TcPOU
FUNCTION_BLOCK CMP_OC_DW
VAR_INPUT
	BOOL_INTERLOCK : BOOL; (*INTERLOCK*)
	DWORD_1: DWORD;		(*WORD 1*)
	END_VAR


VAR_OUTPUT
	BZ_OUTPUT_BOOL : BOOL;
END_VAR


VAR
	OUT_1: BOOL;
END_VAR

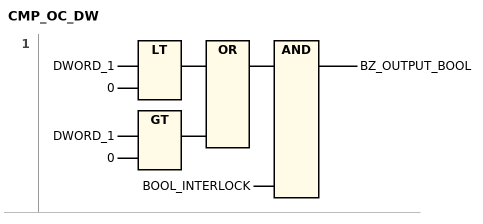
// NETWORK 1
BZ_OUTPUT_BOOL := (DWORD_1 < 0 OR DWORD_1 > 0) AND BOOL_INTERLOCK;

END_FUNCTION_BLOCK

// ---- POUs/MainProgram/AutoArmCtrl/AxisServoCtrl_Arm1.TcPOU
PROGRAM AxisServoCtrl_Arm1
VAR

	fbArm1VertServoMasterController 	: fbV2_ServoMasterController;
	fbArm1HorzServoMasterController 	: fbV2_ServoMasterController;

	iArm1VertStepNumber				: INT;
	iArm1HorzStepNumber				: INT;

	bArm1MCPSOV					: BOOL;
	bArm1MCPSOH					: BOOL;

	bVertDiagBusy					: BOOL;
	bHorzDiagBusy					: BOOL;

	iVertClass3Diag					: INT;
	iHorzClass3Diag					: INT;

	iVertstAX5000C1D					: ST_AX5000_C1D;
	iHorzstAX5000C1D				: ST_AX5000_C1D;

END_VAR

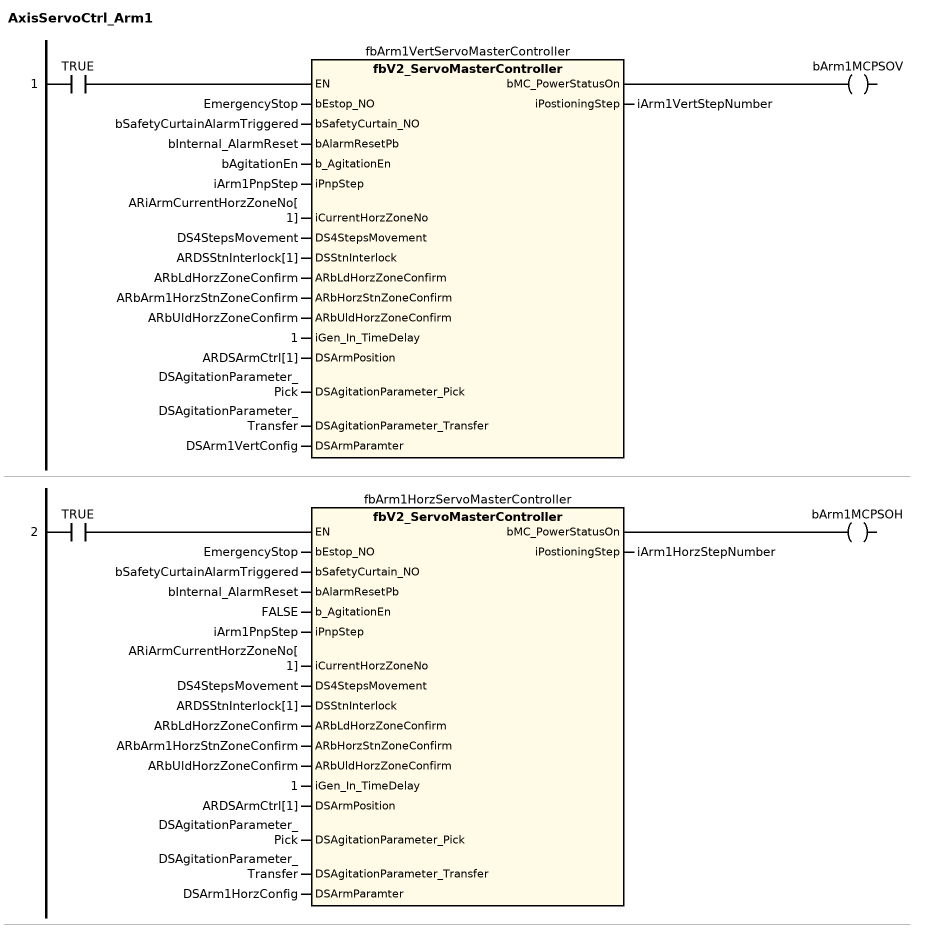
// NETWORK 1
fbArm1VertServoMasterController(
    bEstop_NO := EmergencyStop,
    bSafetyCurtain_NO := bSafetyCurtainAlarmTriggered,
    bAlarmResetPb := bInternal_AlarmReset,
    b_AgitationEn := bAgitationEn,
    iPnpStep := iArm1PnpStep,
    iCurrentHorzZoneNo := ARiArmCurrentHorzZoneNo[1],
    DS4StepsMovement := DS4StepsMovement,
    DSStnInterlock := ARDSStnInterlock[1],
    ARbLdHorzZoneConfirm := ARbLdHorzZoneConfirm,
    ARbHorzStnZoneConfirm := ARbArm1HorzStnZoneConfirm,
    ARbUldHorzZoneConfirm := ARbUldHorzZoneConfirm,
    iGen_In_TimeDelay := 1,
    DSArmPosition := ARDSArmCtrl[1],
    DSAgitationParameter_Pick := DSAgitationParameter_Pick,
    DSAgitationParameter_Transfer := DSAgitationParameter_Transfer,
    DSArmParamter := DSArm1VertConfig,
    iPostioningStep => iArm1VertStepNumber); // fbV2_ServoMasterController
bArm1MCPSOV := fbArm1VertServoMasterController.bMC_PowerStatusOn;

// NETWORK 2
fbArm1HorzServoMasterController(
    bEstop_NO := EmergencyStop,
    bSafetyCurtain_NO := bSafetyCurtainAlarmTriggered,
    bAlarmResetPb := bInternal_AlarmReset,
    b_AgitationEn := FALSE,
    iPnpStep := iArm1PnpStep,
    iCurrentHorzZoneNo := ARiArmCurrentHorzZoneNo[1],
    DS4StepsMovement := DS4StepsMovement,
    DSStnInterlock := ARDSStnInterlock[1],
    ARbLdHorzZoneConfirm := ARbLdHorzZoneConfirm,
    ARbHorzStnZoneConfirm := ARbArm1HorzStnZoneConfirm,
    ARbUldHorzZoneConfirm := ARbUldHorzZoneConfirm,
    iGen_In_TimeDelay := 1,
    DSArmPosition := ARDSArmCtrl[1],
    DSAgitationParameter_Pick := DSAgitationParameter_Pick,
    DSAgitationParameter_Transfer := DSAgitationParameter_Transfer,
    DSArmParamter := DSArm1HorzConfig,
    iPostioningStep => iArm1HorzStepNumber); // fbV2_ServoMasterController
bArm1MCPSOH := fbArm1HorzServoMasterController.bMC_PowerStatusOn;

END_PROGRAM

// ---- POUs/MainProgram/AutoArmCtrl/AxisServoCtrlMapping_Arm1.TcPOU
PROGRAM AxisServoCtrlMapping_Arm1
VAR
	dwArm1Vert4StepsPosBuffer: DWORD;
	dwArm1Vert4StepsPosBufferRE: R_TRIG;

	dwArm1HorzPosBuffer: DWORD;
	dwArm1HorzPosBufferRE: R_TRIG;

	tArm1HorzPosChangeTimer: TON;
	bArm1HorzPosChangeTimerSt: BOOL;

	tArm1Vert4StepPosChangeTimer: TON;
	bArm1Vert4StepPosChangeTimerSt: BOOL;

END_VAR

(*ARM 1*)
IF ARdwVert4StepsPos_In_PositioningEn[1] <> 0 AND ARdwHorzPos_In_PositioningEn[1] = 0 THEN
	ARDSArmCtrl[1].AR3sbTargetPosSt := AR3s_Vert4Steps_bTargetPosSt;
ELSIF ARdwHorzPos_In_PositioningEn[1] <> 0 AND ARdwVert4StepsPos_In_PositioningEn[1] = 0THEN
	ARDSArmCtrl[1].AR3sbTargetPosSt := AR3s_Horz1Step_bTargetPosSt;
ELSE
	ARDSArmCtrl[1].AR3sbTargetPosSt := AR3s_Empty_bTargetPosSt;
END_IF

	bSafetyCurtainAlarmTriggered								:=  ARbDI[eX11011_GeneralSafetyCurtainSensor_Alarm] AND NOT bSafetyDoorSensorBypass ;

(*Home Used*)

(*ARM 1*)

	DSArm1VertConfig.bHome_In_HomingSt							:= dwArm1VertHomeStart <> 0 AND NOT EmergencyStop ;
	DSArm1VertConfig.bHome_In_HomingReset 						:= ( bArmHomeResetbit OR bAutoOriginFE.Q OR bMainOnOffFE.Q OR bMainOnOffRE.Q ) ;
	DSArm1VertConfig.bHome_In_HomeSensor 						:= VertCoERead.bArm1VertHome;
	DSArm1VertConfig.lrHome_In_HighSpeed 						:= ARrArmVertHome1stPercent[1];
	DSArm1VertConfig.lrHome_In_HighSpeedAcc 					:= ARrArmVertHome1stPercentAcc[1];
	DSArm1VertConfig.lrHome_In_HighSpeedDcc 					:= ARrArmVertHome1stPercentDcc[1];
	DSArm1VertConfig.lrHome_In_2ndSpeed 						:= ARrArmVertHome2ndPercent[1];
	DSArm1VertConfig.lrHome_In_2ndSpeedAcc						:= ARrArmVertHome2ndPercentAcc[1];
	DSArm1VertConfig.lrHome_In_2ndSpeedDcc 						:= ARrArmVertHome2ndPercentDcc[1];

	DSArm1VertConfig.rHome_In_DccDelayTimeSec 					:= ARrVertHomeDccDelayTimeSec[1];

	ARbArmVertHomeDone[1]										:= DSArm1VertConfig.bHome_Out_HomeDone ;
	ARbArmVertHomingBusy[1]										:= DSArm1VertConfig.bHome_Out_Busy ;


	DSArm1HorzConfig.bHome_In_HomingSt 							:= (( ARDSArmCtrl[1].AR3sbPositionCfm[2,1,1] AND ARbArmVertHomeDone[1] AND ((ARbArmSlowPullHomeDone[1] AND bArmSlowPulldownCFM) OR bStnLiftoutMechanismBypass) AND NOT EmergencyStop) AND dwArm1HorzHomeStart <> 0 ) ;
	DSArm1HorzConfig.bHome_In_HomingReset 						:= ( bArmHomeResetbit OR bAutoOriginFE.Q OR bMainOnOffFE.Q OR bMainOnOffRE.Q ) ;
	DSArm1HorzConfig.bHome_In_HomeSensor 						:= HorzCoERead.bArm1HorzHome;
	DSArm1HorzConfig.lrHome_In_HighSpeed 						:= ARrArmHorzHome1stPercent[1];
	DSArm1HorzConfig.lrHome_In_HighSpeedAcc 					:= ARrArmHorzHome1stPercentAcc[1];
	DSArm1HorzConfig.lrHome_In_HighSpeedDcc	 					:= ARrArmHorzHome1stPercentDcc[1];
	DSArm1HorzConfig.lrHome_In_2ndSpeed 						:= ARrArmHorzHome2ndPercent[1];
	DSArm1HorzConfig.lrHome_In_2ndSpeedAcc 						:= ARrArmHorzHome2ndPercentAcc[1];
	DSArm1HorzConfig.lrHome_In_2ndSpeedDcc 						:= ARrArmHorzHome2ndPercentDcc[1];

	DSArm1HorzConfig.rHome_In_DccDelayTimeSec 					:= ARrHorzHomeDccDelayTimeSec[1];

	ARbArmHorzHomeDone[1] 										:= DSArm1HorzConfig.bHome_Out_HomeDone ;
	ARbArmHorzHomingBusy[1] 									:= DSArm1HorzConfig.bHome_Out_Busy ;

(*Jog Used*)

(*ARM 1*)

	DSArm1VertConfig.bJog_InOut_JogEn							:= bArmJogEnable (*OR DSV2ApolloRemoteHoistInput.bPB_SelectionSwtich_JogEn*) ;
	DSArm1HorzConfig.bJog_InOut_JogEn                                                		:= bArmJogEnable (*OR DSV2ApolloRemoteHoistInput.bPB_SelectionSwtich_JogEn*) ;

	DSArm1VertConfig.bJog_In_PositiveJogDirectionSt 			:= ARbArmVertJogFwd[1] (*OR ApolloRemoteCtrl.bArmJogDown*);
	DSArm1VertConfig.bJog_In_NegativeJogDirectionSt 			:= ARbArmVertJogRwd[1] (*OR ApolloRemoteCtrl.bArmJogUp*) ;
	DSArm1VertConfig.lrJog_In_JogSpeedHz 						:= ARrArmVertJogPercent[1];
	DSArm1VertConfig.lrJog_In_JogSpeedAcc 						:= ARrArmVertJogAcc[1];
	DSArm1VertConfig.lrJog_In_JogSpeedDcc 						:= ARrArmVertJogDcc[1];

	DSArm1HorzConfig.bJog_In_PositiveJogDirectionSt 			:= ARbArmHorzJogFwd[1] (*OR ApolloRemoteCtrl.bArmJogRight*);
	DSArm1HorzConfig.bJog_In_NegativeJogDirectionSt 			:= ARbArmHorzJogRwd[1] (*OR ApolloRemoteCtrl.bArmJogLeft*);
	DSArm1HorzConfig.lrJog_In_JogSpeedHz 						:= ARrArmHorzJogPercent[1];
	DSArm1HorzConfig.lrJog_In_JogSpeedAcc 						:= ARrArmHorzJogAcc[1];
	DSArm1HorzConfig.lrJog_In_JogSpeedDcc 						:= ARrArmHorzJogDcc[1];

(* Arm Positioning Signal Control Used*)
(* Arm Inv Analog Spd Ctrl Used*)

(*ARM 1*)

	ARbVert_IASC_Out_JogInProgress[1] 							:= DSArm1VertConfig.bOut_JogInProgress;
	ARbVert_IASC_Out_HomeInProgress[1] 							:= DSArm1VertConfig.bOut_HomeInProgress;
	ARbVert_IASC_Out_PosInProgress[1] 							:= DSArm1VertConfig.bOut_PosInProgress ;

	ARbHorz_IASC_Out_JogInProgress[1]  							:= DSArm1HorzConfig.bOut_JogInProgress ;
	ARbHorz_IASC_Out_HomeInProgress[1] 	 						:= DSArm1HorzConfig.bOut_HomeInProgress ;
	ARbHorz_IASC_Out_PosInProgress[1]  							:= DSArm1HorzConfig.bOut_PosInProgress ;


(* General Used*)

(*ARM 1*)

	DSArm1VertConfig.bGen_In_VertMovementEn						:= TRUE;
	DSArm1VertConfig.bGen_In_HorzMovementEn						:= FALSE;

	DSArm1HorzConfig.bGen_In_HorzMovementEn						:= TRUE;
	DSArm1HorzConfig.bGen_In_VertMovementEn						:= FALSE;

	DSArm1VertConfig.bGen_In_FwdOverTravelSensorNC 				:= NOT ARdsEventCtrl[422].bEventOutput ; //Vert Down OT
	DSArm1VertConfig.bGen_In_RwdOverTravelSensorNC 				:= NOT ARdsEventCtrl[421].bEventOutput ; //Vert Up OT

	DSArm1HorzConfig.bGen_In_FwdOverTravelSensorNC 				:= NOT ARdsEventCtrl[425].bEventOutput ; //Horz Uld OT
	DSArm1HorzConfig.bGen_In_RwdOverTravelSensorNC 				:= NOT ARdsEventCtrl[424].bEventOutput ; //Vert Ld OT  


(***********************************************)
(*ARM 1*)
dwArm1HorzPosBufferRE(CLK:= ARdwHorzPos_In_PositioningEn[1] <> dwArm1HorzPosBuffer , Q=> );
IF dwArm1HorzPosBufferRE.Q  THEN
bArm1HorzPosChangeTimerSt := TRUE;
END_IF

tArm1HorzPosChangeTimer(IN:=bArm1HorzPosChangeTimerSt , PT:=t#0.1s , Q=> , ET=> );

IF tArm1HorzPosChangeTimer.Q THEN
dwArm1HorzPosBuffer := ARdwHorzPos_In_PositioningEn[1];
bArm1HorzPosChangeTimerSt := FALSE;
END_IF

(***********************************************)
(***********************************************)
(*ARM 1*)
dwArm1Vert4StepsPosBufferRE(CLK:= ARdwVert4StepsPos_In_PositioningEn[1] <> dwArm1Vert4StepsPosBuffer , Q=> );
IF dwArm1Vert4StepsPosBufferRE.Q THEN
bArm1Vert4StepPosChangeTimerSt := TRUE;
END_IF

tArm1Vert4StepPosChangeTimer(IN:=bArm1Vert4StepPosChangeTimerSt , PT:=t#0.1s , Q=> , ET=> );

IF tArm1Vert4StepPosChangeTimer.Q THEN
dwArm1Vert4StepsPosBuffer := ARdwVert4StepsPos_In_PositioningEn[1];
bArm1Vert4StepPosChangeTimerSt := FALSE;
END_IF

(***********************************************)

(* Pos Ctrl Used*)

(*ARM 1*)

	DSArm1VertConfig.bPos_In_4StepsEn							:= DSArmBasketInfo[1].bAvailibility ;
	DSArm1VertConfig.bPos_In_PositioningEn 						:= ARdwVert4StepsPos_In_PositioningEn[1] <> 0 AND NOT bArm1Vert4StepPosChangeTimerSt ;

	DSArm1VertConfig.lrPos_In_HighSpeed							:= ARlrVertPos_In_HighSpeed[1];
	DSArm1VertConfig.lrPos_In_Acc								:= ARlrVertPos_In_Acc[1];
	DSArm1VertConfig.lrPos_In_Dcc								:= ARlrVertPos_In_Dcc[1];
(*New Added by Lee - 190413*)
	DSArm1VertConfig.bPos_In_Tolerance 							:= 1;

	ARbArmVertMoveDone[1] 										:= DSArm1VertConfig.bPos_Out_PositioningDone;
	ARbArmVertMoveBusy[1] 										:= DSArm1VertConfig.bPos_Out_PositioningBusy ;


	DSArm1HorzConfig.bPos_In_4StepsEn							:= FALSE;
	DSArm1HorzConfig.bPos_In_PositioningEn 						:= ( ARdwHorzPos_In_PositioningEn[1] <> 0 ) AND NOT bArm1HorzPosChangeTimerSt ;

	DSArm1HorzConfig.lrPos_In_HighSpeed							:= ARlrHorzPos_In_HighSpeed[1];
	DSArm1HorzConfig.lrPos_In_Acc								:= ARlrHorzPos_In_Acc[1];
	DSArm1HorzConfig.lrPos_In_Dcc								:= ARlrHorzPos_In_Dcc[1];
(*New Added by Lee - 190413*)
	DSArm1HorzConfig.bPos_In_Tolerance							:= 1;

	ARbArmHorzMoveDone[1] 										:= DSArm1HorzConfig.bPos_Out_PositioningDone ;
	ARbArmHorzMoveBusy[1]  										:= DSArm1HorzConfig.bPos_Out_PositioningBusy ;


	DSArm1VertConfig.bPos_In_Tolerance;
	DSArm1VertConfig.lrGen_Out_CurrentPos;
	DSArm1VertConfig.lrOur_RealTimeSpeedDisplay;
	DSArm1VertConfig.MC_Acc;
	DSArm1VertConfig.MC_ArmContinuosMotion;
	DSArm1VertConfig.MC_ArmDisable;
	DSArm1VertConfig.MC_ArmDiscreteMotion;
	DSArm1VertConfig.MC_ArmErrorStop;
	DSArm1VertConfig.MC_ArmHoming;
	DSArm1VertConfig.MC_ArmStandStill;
	DSArm1VertConfig.MC_ArmStopping;
	DSArm1VertConfig.MC_ArmSynchronizeMotion;
	DSArm1VertConfig.MC_ConstantVelocity;
	DSArm1VertConfig.MC_Dcc;
	
	DSArm1HorzConfig.bPos_In_Tolerance;
	DSArm1HorzConfig.lrGen_Out_CurrentPos;
	DSArm1HorzConfig.lrOur_RealTimeSpeedDisplay;
	DSArm1HorzConfig.MC_Acc;
	DSArm1HorzConfig.MC_ArmContinuosMotion;
	DSArm1HorzConfig.MC_ArmDisable;
	DSArm1HorzConfig.MC_ArmDiscreteMotion;
	DSArm1HorzConfig.MC_ArmErrorStop;
	DSArm1HorzConfig.MC_ArmHoming;
	DSArm1HorzConfig.MC_ArmStandStill;
	DSArm1HorzConfig.MC_ArmStopping;
	DSArm1HorzConfig.MC_ArmSynchronizeMotion;
	DSArm1HorzConfig.MC_ConstantVelocity;
	DSArm1HorzConfig.MC_Dcc;

END_PROGRAM

// ---- POUs/MainProgram/AutoArmCtrl/AxisVertMovementOutputCtrl_Arm1.TcPOU
PROGRAM AxisVertMovementOutputCtrl_Arm1
VAR
	VertTop: CMP_OC_DW;

	LdVertdown: CMP_OC_DW;
	Stn1Vertdown: CMP_OC_DW;
	Stn2Vertdown: CMP_OC_DW;
	Stn3Vertdown: CMP_OC_DW;
	Stn4Vertdown: CMP_OC_DW;
	Stn5Vertdown: CMP_OC_DW;
	Stn6Vertdown: CMP_OC_DW;
	Stn7Vertdown: CMP_OC_DW;
	Stn8Vertdown: CMP_OC_DW;
	Stn9Vertdown: CMP_OC_DW;
	Stn10Vertdown: CMP_OC_DW;
	Stn11Vertdown: CMP_OC_DW;
	Stn12Vertdown: CMP_OC_DW;
	Uld1Vertdown: CMP_OC_DW;
	Uld2Vertdown: CMP_OC_DW;

	Stn8VertSlowPulldown: CMP_OC_DW;

	Stn9VertSlowPulldown: CMP_OC_DW;
END_VAR

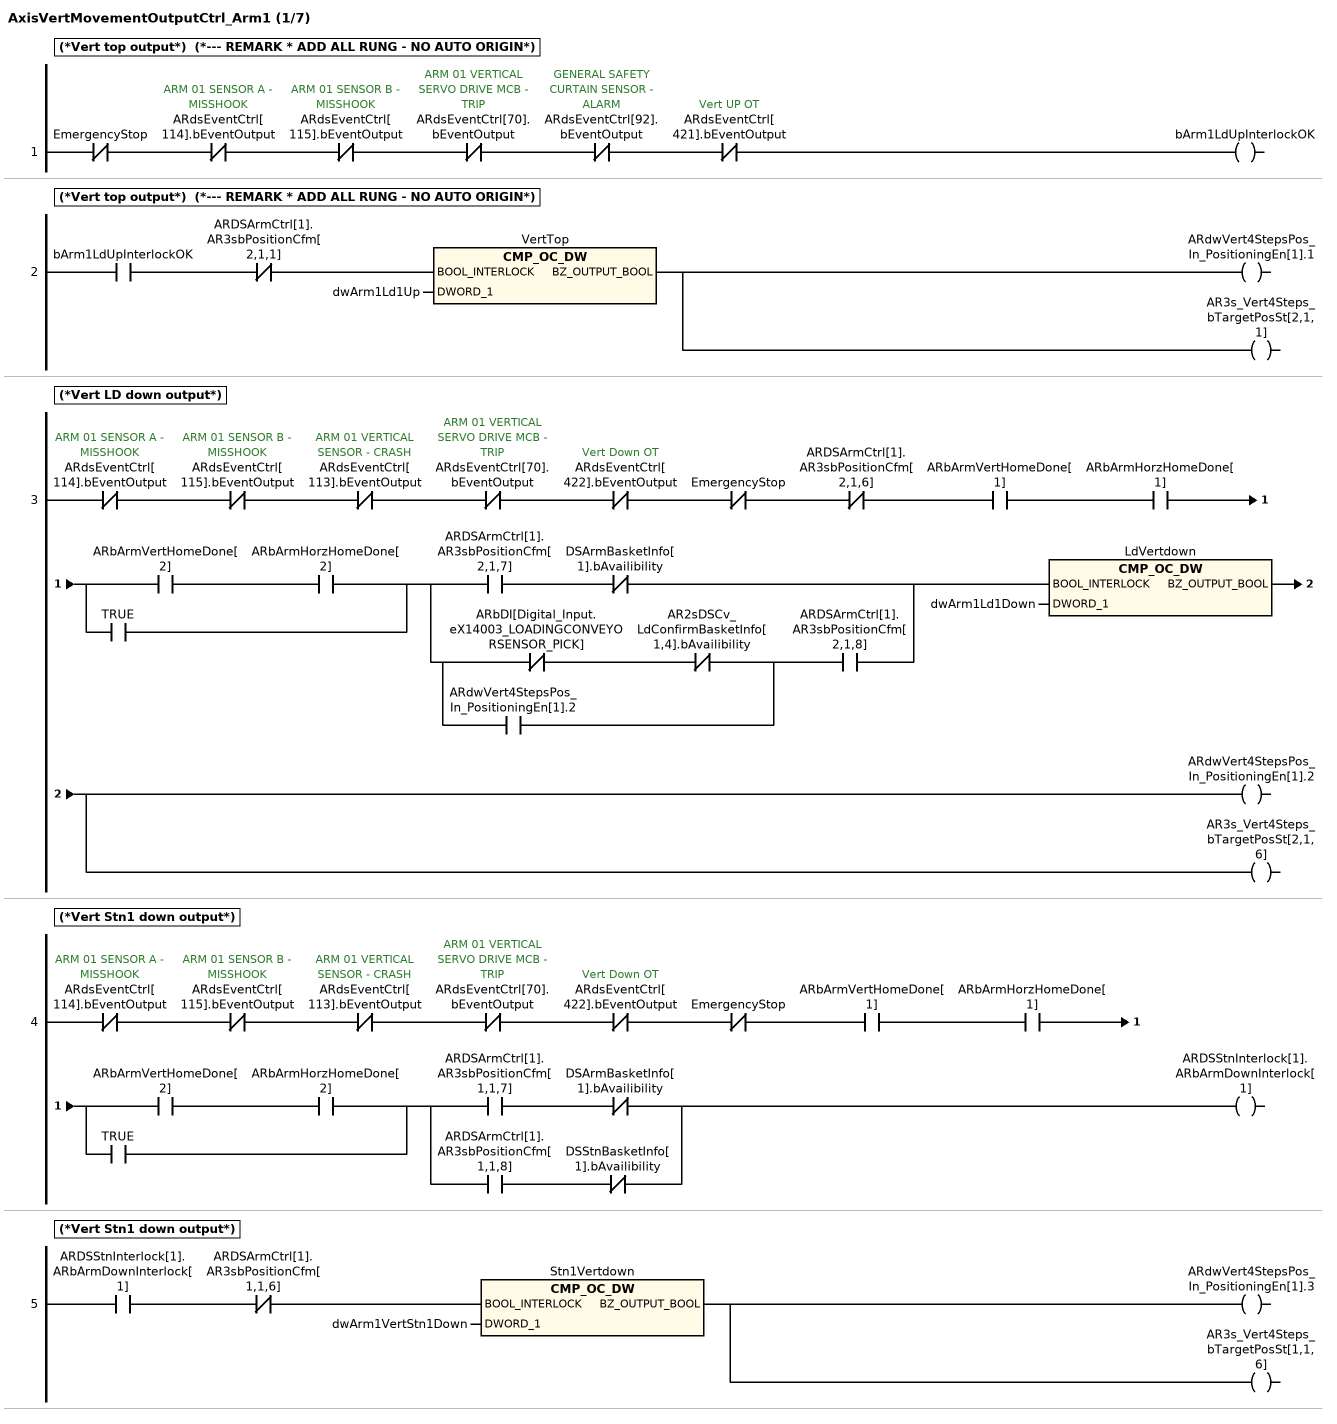
// NETWORK 1
//   ARdsEventCtrl[114].bEventOutput: ARM 01 SENSOR A - MISSHOOK
//   ARdsEventCtrl[115].bEventOutput: ARM 01 SENSOR B - MISSHOOK
//   ARdsEventCtrl[70].bEventOutput: ARM 01 VERTICAL SERVO DRIVE MCB - TRIP
//   ARdsEventCtrl[92].bEventOutput: GENERAL SAFETY CURTAIN SENSOR - ALARM
//   ARdsEventCtrl[421].bEventOutput: Vert UP OT
// label: (*Vert top output*)  (*--- REMARK * ADD ALL RUNG - NO AUTO ORIGIN*)
bArm1LdUpInterlockOK := NOT EmergencyStop AND NOT ARdsEventCtrl[114].bEventOutput AND NOT ARdsEventCtrl[115].bEventOutput AND NOT ARdsEventCtrl[70].bEventOutput AND NOT ARdsEventCtrl[92].bEventOutput AND NOT ARdsEventCtrl[421].bEventOutput;

// NETWORK 2
// label: (*Vert top output*)  (*--- REMARK * ADD ALL RUNG - NO AUTO ORIGIN*)
VertTop(BOOL_INTERLOCK := bArm1LdUpInterlockOK AND NOT ARDSArmCtrl[1].AR3sbPositionCfm[2,1,1], DWORD_1 := dwArm1Ld1Up); // CMP_OC_DW
ARdwVert4StepsPos_In_PositioningEn[1].1 := VertTop.BZ_OUTPUT_BOOL;
AR3s_Vert4Steps_bTargetPosSt[2,1,1] := VertTop.BZ_OUTPUT_BOOL;

// NETWORK 3
//   ARdsEventCtrl[114].bEventOutput: ARM 01 SENSOR A - MISSHOOK
//   ARdsEventCtrl[115].bEventOutput: ARM 01 SENSOR B - MISSHOOK
//   ARdsEventCtrl[113].bEventOutput: ARM 01 VERTICAL SENSOR - CRASH
//   ARdsEventCtrl[70].bEventOutput: ARM 01 VERTICAL SERVO DRIVE MCB - TRIP
//   ARdsEventCtrl[422].bEventOutput: Vert Down OT
// label: (*Vert LD down output*)
LdVertdown(BOOL_INTERLOCK := (NOT ARdsEventCtrl[114].bEventOutput AND NOT ARdsEventCtrl[115].bEventOutput AND NOT ARdsEventCtrl[113].bEventOutput AND NOT ARdsEventCtrl[70].bEventOutput AND NOT ARdsEventCtrl[422].bEventOutput AND NOT EmergencyStop) AND NOT ARDSArmCtrl[1].AR3sbPositionCfm[2,1,6] AND ARbArmVertHomeDone[1] AND ARbArmHorzHomeDone[1] AND (ARbArmVertHomeDone[2] AND ARbArmHorzHomeDone[2] OR TRUE) AND (ARDSArmCtrl[1].AR3sbPositionCfm[2,1,7] AND NOT DSArmBasketInfo[1].bAvailibility OR (NOT ARbDI[Digital_Input.eX14003_LOADINGCONVEYORSENSOR_PICK] AND NOT AR2sDSCv_LdConfirmBasketInfo[1,4].bAvailibility OR ARdwVert4StepsPos_In_PositioningEn[1].2) AND ARDSArmCtrl[1].AR3sbPositionCfm[2,1,8]), DWORD_1 := dwArm1Ld1Down); // CMP_OC_DW
ARdwVert4StepsPos_In_PositioningEn[1].2 := LdVertdown.BZ_OUTPUT_BOOL;
AR3s_Vert4Steps_bTargetPosSt[2,1,6] := LdVertdown.BZ_OUTPUT_BOOL;

// NETWORK 4
//   ARdsEventCtrl[114].bEventOutput: ARM 01 SENSOR A - MISSHOOK
//   ARdsEventCtrl[115].bEventOutput: ARM 01 SENSOR B - MISSHOOK
//   ARdsEventCtrl[113].bEventOutput: ARM 01 VERTICAL SENSOR - CRASH
//   ARdsEventCtrl[70].bEventOutput: ARM 01 VERTICAL SERVO DRIVE MCB - TRIP
//   ARdsEventCtrl[422].bEventOutput: Vert Down OT
// label: (*Vert Stn1 down output*)
ARDSStnInterlock[1].ARbArmDownInterlock[1] := (NOT ARdsEventCtrl[114].bEventOutput AND NOT ARdsEventCtrl[115].bEventOutput AND NOT ARdsEventCtrl[113].bEventOutput AND NOT ARdsEventCtrl[70].bEventOutput AND NOT ARdsEventCtrl[422].bEventOutput AND NOT EmergencyStop) AND ARbArmVertHomeDone[1] AND ARbArmHorzHomeDone[1] AND (ARbArmVertHomeDone[2] AND ARbArmHorzHomeDone[2] OR TRUE) AND (ARDSArmCtrl[1].AR3sbPositionCfm[1,1,7] AND NOT DSArmBasketInfo[1].bAvailibility OR ARDSArmCtrl[1].AR3sbPositionCfm[1,1,8] AND NOT DSStnBasketInfo[1].bAvailibility);

// NETWORK 5
// label: (*Vert Stn1 down output*)
Stn1Vertdown(BOOL_INTERLOCK := ARDSStnInterlock[1].ARbArmDownInterlock[1] AND NOT ARDSArmCtrl[1].AR3sbPositionCfm[1,1,6], DWORD_1 := dwArm1VertStn1Down); // CMP_OC_DW
ARdwVert4StepsPos_In_PositioningEn[1].3 := Stn1Vertdown.BZ_OUTPUT_BOOL;
AR3s_Vert4Steps_bTargetPosSt[1,1,6] := Stn1Vertdown.BZ_OUTPUT_BOOL;

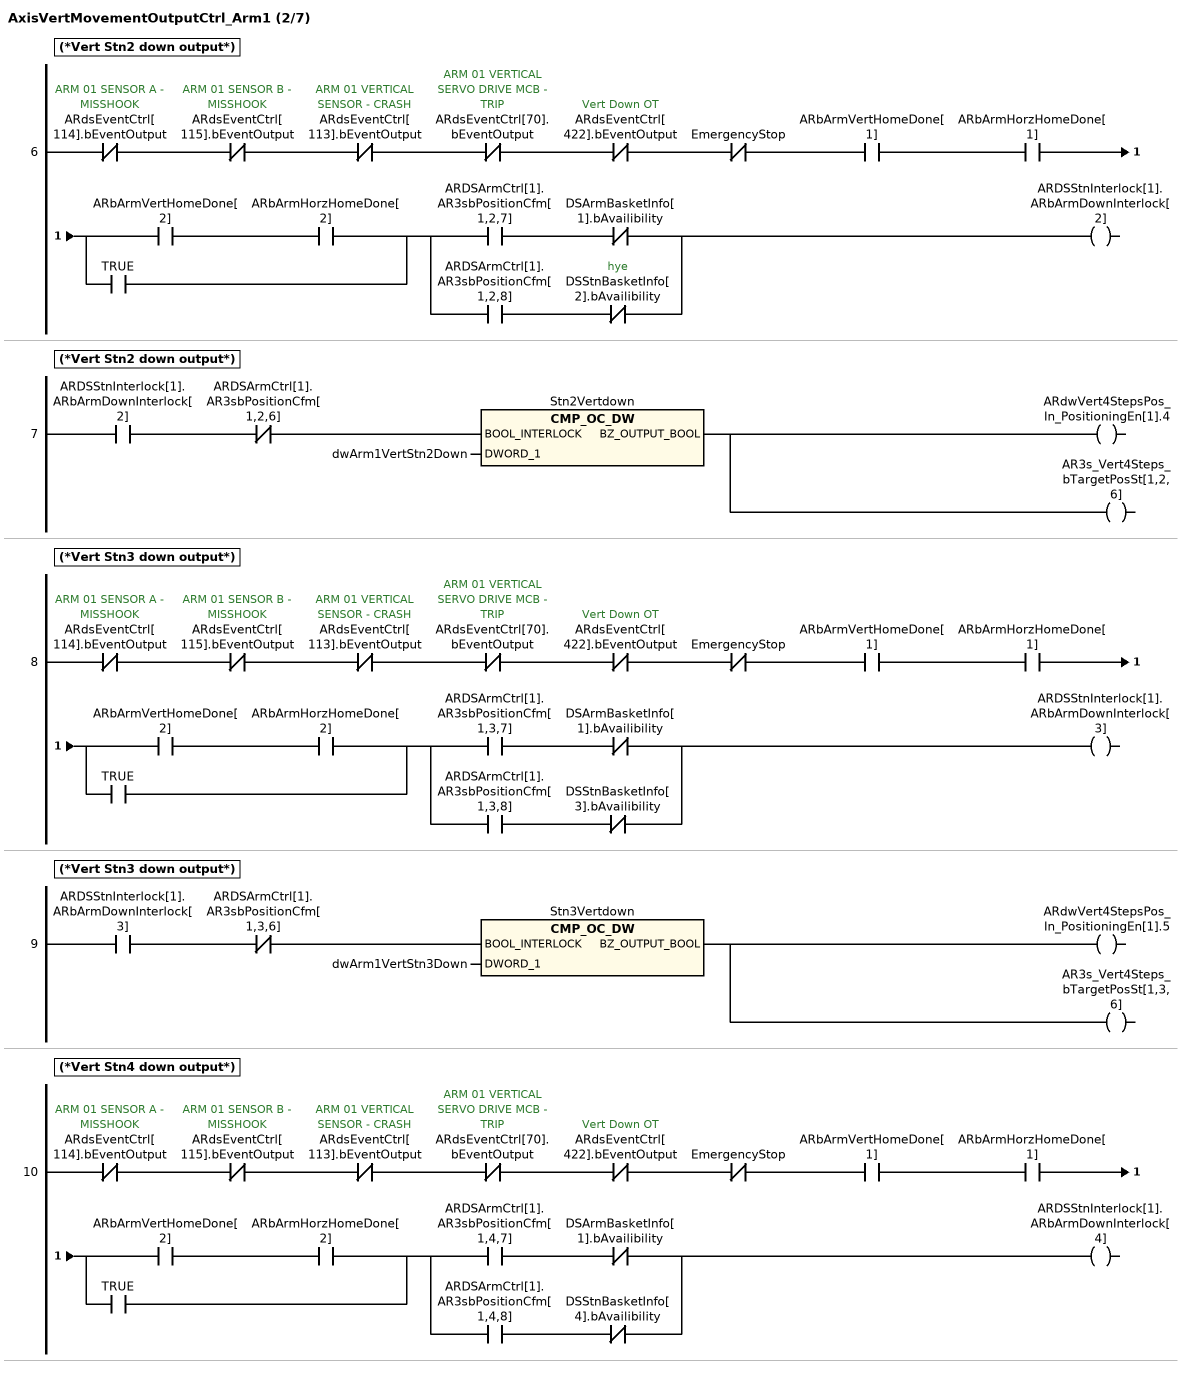
// NETWORK 6
//   ARdsEventCtrl[114].bEventOutput: ARM 01 SENSOR A - MISSHOOK
//   ARdsEventCtrl[115].bEventOutput: ARM 01 SENSOR B - MISSHOOK
//   ARdsEventCtrl[113].bEventOutput: ARM 01 VERTICAL SENSOR - CRASH
//   ARdsEventCtrl[70].bEventOutput: ARM 01 VERTICAL SERVO DRIVE MCB - TRIP
//   ARdsEventCtrl[422].bEventOutput: Vert Down OT
//   DSStnBasketInfo[2].bAvailibility: hye
// label: (*Vert Stn2 down output*)
ARDSStnInterlock[1].ARbArmDownInterlock[2] := (NOT ARdsEventCtrl[114].bEventOutput AND NOT ARdsEventCtrl[115].bEventOutput AND NOT ARdsEventCtrl[113].bEventOutput AND NOT ARdsEventCtrl[70].bEventOutput AND NOT ARdsEventCtrl[422].bEventOutput AND NOT EmergencyStop) AND ARbArmVertHomeDone[1] AND ARbArmHorzHomeDone[1] AND (ARbArmVertHomeDone[2] AND ARbArmHorzHomeDone[2] OR TRUE) AND (ARDSArmCtrl[1].AR3sbPositionCfm[1,2,7] AND NOT DSArmBasketInfo[1].bAvailibility OR ARDSArmCtrl[1].AR3sbPositionCfm[1,2,8] AND NOT DSStnBasketInfo[2].bAvailibility);

// NETWORK 7
// label: (*Vert Stn2 down output*)
Stn2Vertdown(BOOL_INTERLOCK := ARDSStnInterlock[1].ARbArmDownInterlock[2] AND NOT ARDSArmCtrl[1].AR3sbPositionCfm[1,2,6], DWORD_1 := dwArm1VertStn2Down); // CMP_OC_DW
ARdwVert4StepsPos_In_PositioningEn[1].4 := Stn2Vertdown.BZ_OUTPUT_BOOL;
AR3s_Vert4Steps_bTargetPosSt[1,2,6] := Stn2Vertdown.BZ_OUTPUT_BOOL;

// NETWORK 8
//   ARdsEventCtrl[114].bEventOutput: ARM 01 SENSOR A - MISSHOOK
//   ARdsEventCtrl[115].bEventOutput: ARM 01 SENSOR B - MISSHOOK
//   ARdsEventCtrl[113].bEventOutput: ARM 01 VERTICAL SENSOR - CRASH
//   ARdsEventCtrl[70].bEventOutput: ARM 01 VERTICAL SERVO DRIVE MCB - TRIP
//   ARdsEventCtrl[422].bEventOutput: Vert Down OT
// label: (*Vert Stn3 down output*)
ARDSStnInterlock[1].ARbArmDownInterlock[3] := (NOT ARdsEventCtrl[114].bEventOutput AND NOT ARdsEventCtrl[115].bEventOutput AND NOT ARdsEventCtrl[113].bEventOutput AND NOT ARdsEventCtrl[70].bEventOutput AND NOT ARdsEventCtrl[422].bEventOutput AND NOT EmergencyStop) AND ARbArmVertHomeDone[1] AND ARbArmHorzHomeDone[1] AND (ARbArmVertHomeDone[2] AND ARbArmHorzHomeDone[2] OR TRUE) AND (ARDSArmCtrl[1].AR3sbPositionCfm[1,3,7] AND NOT DSArmBasketInfo[1].bAvailibility OR ARDSArmCtrl[1].AR3sbPositionCfm[1,3,8] AND NOT DSStnBasketInfo[3].bAvailibility);

// NETWORK 9
// label: (*Vert Stn3 down output*)
Stn3Vertdown(BOOL_INTERLOCK := ARDSStnInterlock[1].ARbArmDownInterlock[3] AND NOT ARDSArmCtrl[1].AR3sbPositionCfm[1,3,6], DWORD_1 := dwArm1VertStn3Down); // CMP_OC_DW
ARdwVert4StepsPos_In_PositioningEn[1].5 := Stn3Vertdown.BZ_OUTPUT_BOOL;
AR3s_Vert4Steps_bTargetPosSt[1,3,6] := Stn3Vertdown.BZ_OUTPUT_BOOL;

// NETWORK 10
//   ARdsEventCtrl[114].bEventOutput: ARM 01 SENSOR A - MISSHOOK
//   ARdsEventCtrl[115].bEventOutput: ARM 01 SENSOR B - MISSHOOK
//   ARdsEventCtrl[113].bEventOutput: ARM 01 VERTICAL SENSOR - CRASH
//   ARdsEventCtrl[70].bEventOutput: ARM 01 VERTICAL SERVO DRIVE MCB - TRIP
//   ARdsEventCtrl[422].bEventOutput: Vert Down OT
// label: (*Vert Stn4 down output*)
ARDSStnInterlock[1].ARbArmDownInterlock[4] := (NOT ARdsEventCtrl[114].bEventOutput AND NOT ARdsEventCtrl[115].bEventOutput AND NOT ARdsEventCtrl[113].bEventOutput AND NOT ARdsEventCtrl[70].bEventOutput AND NOT ARdsEventCtrl[422].bEventOutput AND NOT EmergencyStop) AND ARbArmVertHomeDone[1] AND ARbArmHorzHomeDone[1] AND (ARbArmVertHomeDone[2] AND ARbArmHorzHomeDone[2] OR TRUE) AND (ARDSArmCtrl[1].AR3sbPositionCfm[1,4,7] AND NOT DSArmBasketInfo[1].bAvailibility OR ARDSArmCtrl[1].AR3sbPositionCfm[1,4,8] AND NOT DSStnBasketInfo[4].bAvailibility);

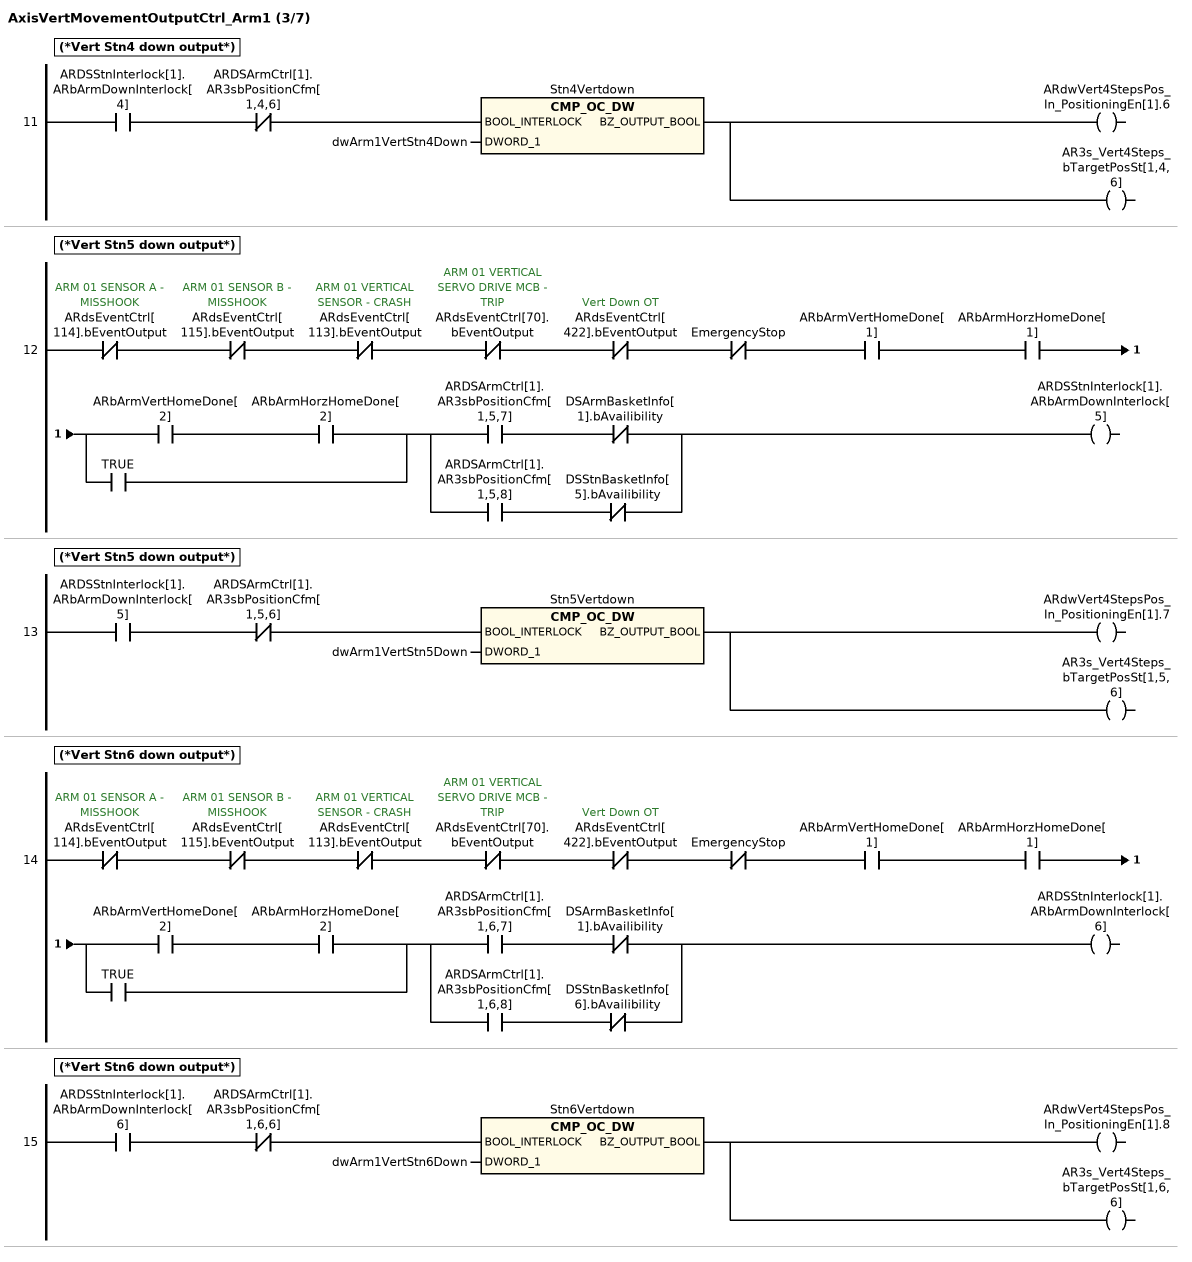
// NETWORK 11
// label: (*Vert Stn4 down output*)
Stn4Vertdown(BOOL_INTERLOCK := ARDSStnInterlock[1].ARbArmDownInterlock[4] AND NOT ARDSArmCtrl[1].AR3sbPositionCfm[1,4,6], DWORD_1 := dwArm1VertStn4Down); // CMP_OC_DW
ARdwVert4StepsPos_In_PositioningEn[1].6 := Stn4Vertdown.BZ_OUTPUT_BOOL;
AR3s_Vert4Steps_bTargetPosSt[1,4,6] := Stn4Vertdown.BZ_OUTPUT_BOOL;

// NETWORK 12
//   ARdsEventCtrl[114].bEventOutput: ARM 01 SENSOR A - MISSHOOK
//   ARdsEventCtrl[115].bEventOutput: ARM 01 SENSOR B - MISSHOOK
//   ARdsEventCtrl[113].bEventOutput: ARM 01 VERTICAL SENSOR - CRASH
//   ARdsEventCtrl[70].bEventOutput: ARM 01 VERTICAL SERVO DRIVE MCB - TRIP
//   ARdsEventCtrl[422].bEventOutput: Vert Down OT
// label: (*Vert Stn5 down output*)
ARDSStnInterlock[1].ARbArmDownInterlock[5] := (NOT ARdsEventCtrl[114].bEventOutput AND NOT ARdsEventCtrl[115].bEventOutput AND NOT ARdsEventCtrl[113].bEventOutput AND NOT ARdsEventCtrl[70].bEventOutput AND NOT ARdsEventCtrl[422].bEventOutput AND NOT EmergencyStop) AND ARbArmVertHomeDone[1] AND ARbArmHorzHomeDone[1] AND (ARbArmVertHomeDone[2] AND ARbArmHorzHomeDone[2] OR TRUE) AND (ARDSArmCtrl[1].AR3sbPositionCfm[1,5,7] AND NOT DSArmBasketInfo[1].bAvailibility OR ARDSArmCtrl[1].AR3sbPositionCfm[1,5,8] AND NOT DSStnBasketInfo[5].bAvailibility);

// NETWORK 13
// label: (*Vert Stn5 down output*)
Stn5Vertdown(BOOL_INTERLOCK := ARDSStnInterlock[1].ARbArmDownInterlock[5] AND NOT ARDSArmCtrl[1].AR3sbPositionCfm[1,5,6], DWORD_1 := dwArm1VertStn5Down); // CMP_OC_DW
ARdwVert4StepsPos_In_PositioningEn[1].7 := Stn5Vertdown.BZ_OUTPUT_BOOL;
AR3s_Vert4Steps_bTargetPosSt[1,5,6] := Stn5Vertdown.BZ_OUTPUT_BOOL;

// NETWORK 14
//   ARdsEventCtrl[114].bEventOutput: ARM 01 SENSOR A - MISSHOOK
//   ARdsEventCtrl[115].bEventOutput: ARM 01 SENSOR B - MISSHOOK
//   ARdsEventCtrl[113].bEventOutput: ARM 01 VERTICAL SENSOR - CRASH
//   ARdsEventCtrl[70].bEventOutput: ARM 01 VERTICAL SERVO DRIVE MCB - TRIP
//   ARdsEventCtrl[422].bEventOutput: Vert Down OT
// label: (*Vert Stn6 down output*)
ARDSStnInterlock[1].ARbArmDownInterlock[6] := (NOT ARdsEventCtrl[114].bEventOutput AND NOT ARdsEventCtrl[115].bEventOutput AND NOT ARdsEventCtrl[113].bEventOutput AND NOT ARdsEventCtrl[70].bEventOutput AND NOT ARdsEventCtrl[422].bEventOutput AND NOT EmergencyStop) AND ARbArmVertHomeDone[1] AND ARbArmHorzHomeDone[1] AND (ARbArmVertHomeDone[2] AND ARbArmHorzHomeDone[2] OR TRUE) AND (ARDSArmCtrl[1].AR3sbPositionCfm[1,6,7] AND NOT DSArmBasketInfo[1].bAvailibility OR ARDSArmCtrl[1].AR3sbPositionCfm[1,6,8] AND NOT DSStnBasketInfo[6].bAvailibility);

// NETWORK 15
// label: (*Vert Stn6 down output*)
Stn6Vertdown(BOOL_INTERLOCK := ARDSStnInterlock[1].ARbArmDownInterlock[6] AND NOT ARDSArmCtrl[1].AR3sbPositionCfm[1,6,6], DWORD_1 := dwArm1VertStn6Down); // CMP_OC_DW
ARdwVert4StepsPos_In_PositioningEn[1].8 := Stn6Vertdown.BZ_OUTPUT_BOOL;
AR3s_Vert4Steps_bTargetPosSt[1,6,6] := Stn6Vertdown.BZ_OUTPUT_BOOL;

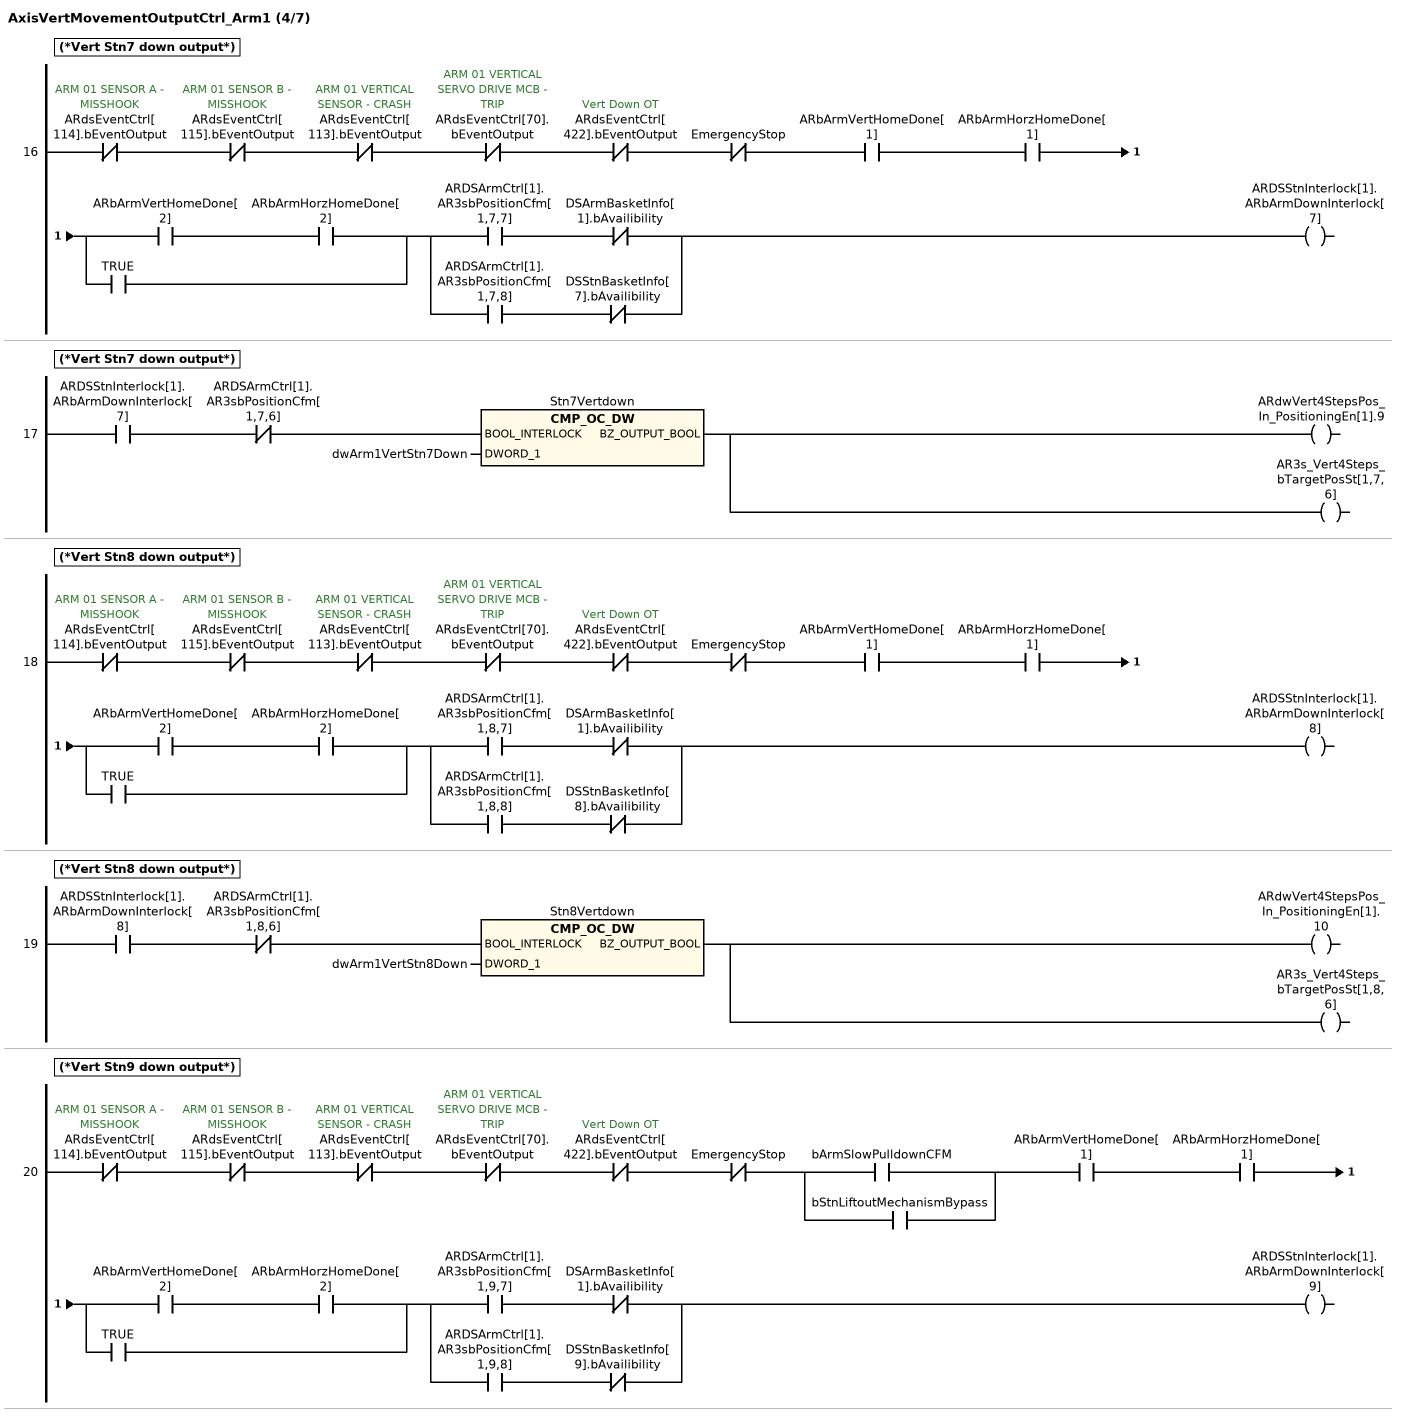
// NETWORK 16
//   ARdsEventCtrl[114].bEventOutput: ARM 01 SENSOR A - MISSHOOK
//   ARdsEventCtrl[115].bEventOutput: ARM 01 SENSOR B - MISSHOOK
//   ARdsEventCtrl[113].bEventOutput: ARM 01 VERTICAL SENSOR - CRASH
//   ARdsEventCtrl[70].bEventOutput: ARM 01 VERTICAL SERVO DRIVE MCB - TRIP
//   ARdsEventCtrl[422].bEventOutput: Vert Down OT
// label: (*Vert Stn7 down output*)
ARDSStnInterlock[1].ARbArmDownInterlock[7] := (NOT ARdsEventCtrl[114].bEventOutput AND NOT ARdsEventCtrl[115].bEventOutput AND NOT ARdsEventCtrl[113].bEventOutput AND NOT ARdsEventCtrl[70].bEventOutput AND NOT ARdsEventCtrl[422].bEventOutput AND NOT EmergencyStop) AND ARbArmVertHomeDone[1] AND ARbArmHorzHomeDone[1] AND (ARbArmVertHomeDone[2] AND ARbArmHorzHomeDone[2] OR TRUE) AND (ARDSArmCtrl[1].AR3sbPositionCfm[1,7,7] AND NOT DSArmBasketInfo[1].bAvailibility OR ARDSArmCtrl[1].AR3sbPositionCfm[1,7,8] AND NOT DSStnBasketInfo[7].bAvailibility);

// NETWORK 17
// label: (*Vert Stn7 down output*)
Stn7Vertdown(BOOL_INTERLOCK := ARDSStnInterlock[1].ARbArmDownInterlock[7] AND NOT ARDSArmCtrl[1].AR3sbPositionCfm[1,7,6], DWORD_1 := dwArm1VertStn7Down); // CMP_OC_DW
ARdwVert4StepsPos_In_PositioningEn[1].9 := Stn7Vertdown.BZ_OUTPUT_BOOL;
AR3s_Vert4Steps_bTargetPosSt[1,7,6] := Stn7Vertdown.BZ_OUTPUT_BOOL;

// NETWORK 18
//   ARdsEventCtrl[114].bEventOutput: ARM 01 SENSOR A - MISSHOOK
//   ARdsEventCtrl[115].bEventOutput: ARM 01 SENSOR B - MISSHOOK
//   ARdsEventCtrl[113].bEventOutput: ARM 01 VERTICAL SENSOR - CRASH
//   ARdsEventCtrl[70].bEventOutput: ARM 01 VERTICAL SERVO DRIVE MCB - TRIP
//   ARdsEventCtrl[422].bEventOutput: Vert Down OT
// label: (*Vert Stn8 down output*)
ARDSStnInterlock[1].ARbArmDownInterlock[8] := (NOT ARdsEventCtrl[114].bEventOutput AND NOT ARdsEventCtrl[115].bEventOutput AND NOT ARdsEventCtrl[113].bEventOutput AND NOT ARdsEventCtrl[70].bEventOutput AND NOT ARdsEventCtrl[422].bEventOutput AND NOT EmergencyStop) AND ARbArmVertHomeDone[1] AND ARbArmHorzHomeDone[1] AND (ARbArmVertHomeDone[2] AND ARbArmHorzHomeDone[2] OR TRUE) AND (ARDSArmCtrl[1].AR3sbPositionCfm[1,8,7] AND NOT DSArmBasketInfo[1].bAvailibility OR ARDSArmCtrl[1].AR3sbPositionCfm[1,8,8] AND NOT DSStnBasketInfo[8].bAvailibility);

// NETWORK 19
// label: (*Vert Stn8 down output*)
Stn8Vertdown(BOOL_INTERLOCK := ARDSStnInterlock[1].ARbArmDownInterlock[8] AND NOT ARDSArmCtrl[1].AR3sbPositionCfm[1,8,6], DWORD_1 := dwArm1VertStn8Down); // CMP_OC_DW
ARdwVert4StepsPos_In_PositioningEn[1].10 := Stn8Vertdown.BZ_OUTPUT_BOOL;
AR3s_Vert4Steps_bTargetPosSt[1,8,6] := Stn8Vertdown.BZ_OUTPUT_BOOL;

// NETWORK 20
//   ARdsEventCtrl[114].bEventOutput: ARM 01 SENSOR A - MISSHOOK
//   ARdsEventCtrl[115].bEventOutput: ARM 01 SENSOR B - MISSHOOK
//   ARdsEventCtrl[113].bEventOutput: ARM 01 VERTICAL SENSOR - CRASH
//   ARdsEventCtrl[70].bEventOutput: ARM 01 VERTICAL SERVO DRIVE MCB - TRIP
//   ARdsEventCtrl[422].bEventOutput: Vert Down OT
// label: (*Vert Stn9 down output*)
ARDSStnInterlock[1].ARbArmDownInterlock[9] := (NOT ARdsEventCtrl[114].bEventOutput AND NOT ARdsEventCtrl[115].bEventOutput AND NOT ARdsEventCtrl[113].bEventOutput AND NOT ARdsEventCtrl[70].bEventOutput AND NOT ARdsEventCtrl[422].bEventOutput AND NOT EmergencyStop AND (bArmSlowPulldownCFM OR bStnLiftoutMechanismBypass)) AND ARbArmVertHomeDone[1] AND ARbArmHorzHomeDone[1] AND (ARbArmVertHomeDone[2] AND ARbArmHorzHomeDone[2] OR TRUE) AND (ARDSArmCtrl[1].AR3sbPositionCfm[1,9,7] AND NOT DSArmBasketInfo[1].bAvailibility OR ARDSArmCtrl[1].AR3sbPositionCfm[1,9,8] AND NOT DSStnBasketInfo[9].bAvailibility);

